screen "Root screen" 800x480, template "Main"
   Button "Button_1" at 525,223 size 98x74; TextOff 'Text'
      on Click: InvertBit("V1_CMD_Start_M")
      Visibility <- "Logick_hand"
   Button "Button_2" at 409,219 size 32x177; TextOff 'Text'
      on Click: InvertBit("V2_CMD_Start_M")
      Visibility <- "Logick_hand"
   Button "Button_6" at 252,16 size 115x197; TextOff 'Text'
      on Click: InvertBit("T1_CMD_Start_M")
      Visibility <- "Logick_hand"
   Button "Button_12" at 225,303 size 168x65; TextOff 'Text'
      on Click: InvertBit("T3_CMD_Start_M")
      Visibility <- "Logick_hand"
   Button "Button_13" at 453,307 size 192x61; TextOff 'Text'
      on Click: InvertBit("T2_CMD_Start_M")
      Visibility <- "Logick_hand"
   Button "Button_3" at 269,227 size 85x72; TextOff 'Text'
      on Click: InvertBit("V3_CMD_Start_M")
      Visibility <- "Logick_hand"
   Button "Button_4" at 175,16 size 73x115; TextOff 'Text'
      on Click: InvertBit("T0_CMD_Start_M")
      Visibility <- "Logick_hand"
   Rectangle "Rectangle_25" at 421,348 size 10x46
      Visibility <- "Valves_DB_V2_Status"
   IOField "I/O field_1" at 262,49 size 96x32; FormatPattern 999.9
      ProcessValue <- "AOx_DB_SP_CF_SP_M"
      Appearance <- "AOx_DB_SP_CF_CMD_Hand"
   Rectangle "Rectangle_17" at 130,379 size 23x10
      Appearance <- "T3_Box_Ready_Signal"
   Rectangle "Rectangle_18" at 133,375 size 17x5
      Appearance <- "T3_Box_Ready_Signal"
   Rectangle "Rectangle_19" at 302,379 size 23x10
      Appearance <- "T2_Box_Ready_Signal"
   Rectangle "Rectangle_20" at 305,375 size 17x5
      Appearance <- "T2_Box_Ready_Signal"
   Rectangle "Rectangle_21" at 451,379 size 23x10
      Appearance <- "T1_Box_ready_Signal"
   Rectangle "Rectangle_22" at 454,375 size 17x5
      Appearance <- "T1_Box_ready_Signal"
   Button "Button_15" at 31,168 size 178x54; TextOff 'Пропустить'
      on Click: SetBit("T3V3W3_DB_Skip_box")
      Appearance <- "main_screens"
   Rectangle "Rectangle_2" at 252,16 size 115x230
      Appearance <- "T1_Status"
   Rectangle "Rectangle_3" at 14,253 size 199x115
      Appearance <- "T4_Status"
   Rectangle "Rectangle_4" at 225,253 size 168x115
      Appearance <- "T3_Status"
   Rectangle "Rectangle_5" at 406,253 size 239x115
      Appearance <- "T2_Status"
   Rectangle "Rectangle_6" at 421,247 size 10x46
      Visibility <- "Valves_DB_V2_Status"
   Rectangle "Rectangle_7" at 421,326 size 10x46
      Visibility <- "Valves_DB_V2_Status"
   Rectangle "Rectangle_8" at 568,243 size 10x38
      Visibility <- "Valves_DB_V1_Status"
   Rectangle "Rectangle_9" at 542,280 size 62x10
      Visibility <- "Valves_DB_V1_Status"
   TextField "Text field_2" at 612,341 size 49x28; Text 'T2'
   TextField "Text field_3" at 361,340 size 49x28; Text 'T3'
   TextField "Text field_4" at 178,341 size 49x28; Text 'T4'
   Rectangle "Rectangle_10" at 421,223 size 10x46
      Visibility <- "Valves_DB_V2_Status"
   Rectangle "Rectangle_11" at 421,348 size 10x46
      Visibility <- "Valves_DB_V2_Status"
   Rectangle "Rectangle_12" at 569,223 size 10x38
      Visibility <- "Valves_DB_V1_Status"
   Rectangle "Rectangle_13" at 543,260 size 62x10
      Visibility <- "Valves_DB_V1_Status"
   TextField "Text field_7" at 433,227 size 43x23; Text 'V2'
   TextField "Text field_8" at 579,227 size 43x23; Text 'V1'
   Button "Button_8" at 376,17 size 175x60; TextOff 'Авто'
      on Release: SetBit("Logic_DB_Start_weight")
      Appearance <- "Logic_DB_Start_weight"
   Button "Button_9" at 376,85 size 175x60; TextOff 'Стоп'
      on Release: ResetBit("Logic_DB_Start_weight")
   Button "Button_10" at 376,153 size 175x60; TextOff 'Ручной'; Authorization "Operator"
      on Click: InvertBit("Logick_hand")
      Appearance <- "Logick_hand"
   IOField "I/O field_4" at 556,17 size 175x60; FormatPattern 99.9
      ProcessValue <- "T3V3W3_DB_SetPoints_SP"
   TextField "Text field_17" at 588,84 size 112x62; Text 'кг'
   Rectangle "Rectangle_24" at 421,223 size 10x46
      Visibility <- "Valves_DB_V2_Status"
   Rectangle "Rectangle_26" at 421,223 size 10x46
      Visibility <- "Valves_DB_V2_Status"
   Rectangle "Rectangle_27" at 421,348 size 10x46
      Visibility <- "Valves_DB_V2_Status"
   Rectangle "Rectangle_28" at 569,224 size 10x38
      Visibility <- "Valves_DB_V1_Status"
   Rectangle "Rectangle_29" at 543,260 size 62x10
      Visibility <- "Valves_DB_V1_Status"
   Rectangle "Rectangle_30" at 569,224 size 10x38
      Visibility <- "Valves_DB_V1_Status"
   Rectangle "Rectangle_31" at 543,260 size 62x10
      Visibility <- "Valves_DB_V1_Status"
   TextField "Text field_11" at 20,48 size 135x52; Text 'Тунель охлаждения'
   IOField "I/O field_2" at 556,153 size 175x60; FormatPattern s99.9
      ProcessValue <- "T3V3W3_DB_LocalVar_SP_loaded"
   Rectangle "Rectangle_32" at 175,16 size 73x115
      Appearance <- "T0_Status"
   TextField "Text field_1" at 189,15 size 49x28; Text 'T0'
   TextField "Text field_12" at 285,13 size 49x28; Text 'T1'
   Circle "Circle_1" at 270,220 size 82x82
      Appearance <- "V3_Status"
   Button "Button_11" at 14,253 size 199x115; TextOff 'Text'
      on Click: InvertBit("T4_CMD_Start_M")
      Visibility <- "Logick_hand"
   TextField "Text field_13" at 298,250 size 43x23; Text 'V3'
   Group "Group" at 130,375 size 23x30
   Group "Group_1" at 302,375 size 23x30
   Group "Group_2" at 451,375 size 23x30
   TextField "Template_Text field_1" at 525,59 size 27x15; Text 'F1'
   TextField "Template_Text field_2" at 525,127 size 27x15; Text 'F2'
   Button "Button_21" at 556,153 size 173x61; TextOff 'Установка нуля'; TextList "Hand"
      on Click: InvertBit("T3V3W3_DB_Reset_weight")
      ProcessValue <- "ODT1_CMD_Hand"
      Visibility <- "Logic_DB_Start_weight"
   Button "Button_5" at 14,415 size 211x58; TextOff 'Обзор'
      on Click: ActivateScreen("Root screen", 0); SetTag("main_screens", 0)
      Appearance <- "main_screens"
   Button "Button_14" at 264,415 size 211x58; TextOff 'Вес'
      on Click: ActivateScreen("weight", 0); SetTag("main_screens", 1)
      Appearance <- "main_screens"
   Button "Button_7" at 513,415 size 211x58; TextOff 'Статистика'
      on Click: ActivateScreen("statistic", 0); SetTag("main_screens", 2); SetTag("stat_view", 0)
      Appearance <- "main_screens"
   Rectangle "Rectangle_33" at 5,269 size 732x211
      Visibility <- "T3V3W3_DB_Reload"
   Rectangle "Rectangle_23" at 32,134 size 175x115
      Visibility <- "Any_Hand"
      Appearance <- "Any_Hand"
   TextField "Text field_5" at 142,306 size 455x58; Text 'Некорректный вес.'
      Visibility <- "T3V3W3_DB_Reload"
   Button "Button_16" at 193,388 size 345x75; TextOff 'Продолжить'
      on Click: SetBit("Reset_All")
      Visibility <- "T3V3W3_DB_Reload"
   TextField "Text field_10" at 36,140 size 169x99; Text 'Внимание! Часть устройств в ручном режиме. Корректная работа невозможна.'
      Visibility <- "Any_Hand"
      Appearance <- "Any_Hand"
   Rectangle "Rectangle_34" at 5,268 size 732x211
      Visibility <- "T3V3W3_DB_No_box"
   Button "Button_20" at 197,387 size 345x75; TextOff 'Продолжить'
      on Click: ResetBit("T3V3W3_DB_No_box")
      Visibility <- "T3V3W3_DB_No_box"
   TextField "Text field_6" at 216,305 size 311x58; Text 'Нет коробки.'
      Visibility <- "T3V3W3_DB_No_box"

screen "Conveyors_0" 800x480, template "Main"
   Rectangle "Rectangle_2" at 127,146 size 416x126
      Appearance <- "T3_CMD_Sim"
   GraphicIOField "Graphic I/O field_1" at 134,182 size 43x85; PictureList "Motor"
      ProcessValue <- "T3_Status"
   Button "Button_10" at 213,180 size 90x22; TextOff 'Авто'; TextList "Hand"
      on Click: InvertBit("T3_CMD_Hand")
      Appearance <- "T3_CMD_Hand"
      ProcessValue <- "T3_CMD_Hand"
   Button "Button_12" at 258,202 size 45x22; TextOff 'Выкл'
      on Click: ResetBit("T3_CMD_Start_M")
   Button "Button_14" at 213,225 size 90x20; TextOff 'Сервис'
      on Click: InvertBit("T3_CMD_Service")
      Appearance <- "T3_CMD_Service"
   Button "Button_15" at 213,202 size 45x22; TextOff 'Вкл'
      on Click: SetBit("T3_CMD_Start_M")
      Appearance <- "T3_CMD_Start_M"
   TextField "Text field_6" at 133,151 size 171x26; Text 'Конвеер 3'
   TextField "Text field_7" at 310,151 size 99x18; Text 'Ожидание ОС, с'
   GraphicView "Graphic view_2" at 180,181 size 25x25; Picture "z2use_3"
      Visibility <- "T3_CMD_Hand"
   GraphicView "Graphic view_3" at 180,213 size 25x25; Picture "force"
      Visibility <- "T3_CMD_Force"
   GraphicView "Graphic view_4" at 180,242 size 25x25; Picture "service"
      Visibility <- "T3_CMD_Service"
   TextField "Text field_8" at 436,170 size 20x18; Text 'QF'
   TextField "Text field_9" at 436,195 size 21x18; Text 'KM'
   TextField "Text field_11" at 436,221 size 44x18; Text 'Service'
   TextField "Text field_16" at 436,247 size 41x18; Text 'Termo'
   TextField "Text field_17" at 416,149 size 120x22; Text 'Использовать:'
   Button "Button_16" at 478,171 size 60x20; TextOff 'Text'; PictureList "ON_OFF"; Authorization "Operator"
      on Click: InvertBit("T3_Use_QF")
      ProcessValue <- "T3_Use_QF"
   Button "Button_17" at 478,195 size 60x20; TextOff 'Text'; Authorization "Operator"; PictureList "ON_OFF"
      on Click: InvertBit("T3_Use_KM")
      ProcessValue <- "T3_Use_KM"
   Button "Button_18" at 478,219 size 60x20; TextOff 'Text'; Authorization "Operator"; PictureList "ON_OFF"
      on Click: InvertBit("T3_Use_Serivce")
      ProcessValue <- "T3_Use_Serivce"
   Button "Button_19" at 478,244 size 60x20; TextOff 'Text'; Authorization "Operator"; PictureList "ON_OFF"
      on Click: InvertBit("T3_Use_Termo")
      ProcessValue <- "T3_Use_Termo"
   Button "Button_20" at 416,170 size 20x20; TextOff 'Text'; PictureList "ok"; Authorization "Operator"
      ProcessValue <- "T3_FB_QF"
   Button "Button_23" at 416,194 size 20x20; TextOff 'Text'; Authorization "Operator"; PictureList "ok"
      ProcessValue <- "T3_FB_KM"
   Button "Button_28" at 416,219 size 20x20; TextOff 'Text'; Authorization "Operator"; PictureList "ok"
      ProcessValue <- "T3_Use_Serivce"
   Button "Button_31" at 416,244 size 20x20; TextOff 'Text'; Authorization "Operator"; PictureList "ok"
      ProcessValue <- "T3_FB_Termo"
   TextField "Text field_18" at 323,226 size 79x18; Text 'Наработка, ч'
   TextField "Text field_19" at 309,173 size 37x18; Text 'Старт'
   IOField "I/O field_1" at 348,171 size 30x20; FormatPattern 99
      ProcessValue <- "T3_Wait_On_SP"
   IOField "I/O field_2" at 348,194 size 30x20; FormatPattern 99
      ProcessValue <- "T3_Wait_Off_SP"
   TextField "Text field_20" at 309,194 size 32x18; Text 'Стоп'
   IOField "I/O field_3" at 378,171 size 30x20; FormatPattern 99
      ProcessValue <- "T3_Wait_On_Now"
   IOField "I/O field_4" at 378,194 size 30x20; FormatPattern 99
      ProcessValue <- "T3_Wait_Off_Now"
   IOField "I/O field_6" at 313,244 size 98x20; FormatPattern 9999999999
      ProcessValue <- "T3_Res_h"
   Button "Button_32" at 213,245 size 90x20; TextOff 'Force'
      on Click: InvertBit("T3_CMD_Force")
      Appearance <- "T3_CMD_Force"
   Rectangle "Rectangle_3" at 127,285 size 416x126
      Appearance <- "T4_CMD_Sim"
   GraphicIOField "Graphic I/O field_3" at 134,321 size 43x85; PictureList "Motor"
      ProcessValue <- "T4_Status"
   Button "Button_33" at 213,319 size 90x22; TextOff 'Авто'; TextList "Hand"
      on Click: InvertBit("T4_CMD_Hand")
      Appearance <- "T4_CMD_Hand"
      ProcessValue <- "T4_CMD_Hand"
   Button "Button_34" at 258,341 size 45x22; TextOff 'Выкл'
      on Click: ResetBit("T4_CMD_Start_M")
   Button "Button_35" at 213,364 size 90x20; TextOff 'Сервис'
      on Click: InvertBit("T4_CMD_Service")
      Appearance <- "T4_CMD_Service"
   Button "Button_36" at 213,341 size 45x22; TextOff 'Вкл'
      on Click: SetBit("T4_CMD_Start_M")
      Appearance <- "T4_CMD_Start_M"
   TextField "Text field_21" at 133,290 size 171x26; Text 'Конвеер 4'
   TextField "Text field_22" at 310,290 size 99x18; Text 'Ожидание ОС, с'
   GraphicView "Graphic view_5" at 180,320 size 25x25; Picture "z2use_3"
      Visibility <- "T4_CMD_Hand"
   GraphicView "Graphic view_6" at 180,352 size 25x25; Picture "force"
      Visibility <- "T4_CMD_Force"
   GraphicView "Graphic view_7" at 180,381 size 25x25; Picture "service"
      Visibility <- "T4_CMD_Service"
   TextField "Text field_23" at 436,309 size 20x18; Text 'QF'
   TextField "Text field_24" at 436,334 size 21x18; Text 'KM'
   TextField "Text field_25" at 436,360 size 44x18; Text 'Service'
   TextField "Text field_26" at 436,386 size 41x18; Text 'Termo'
   TextField "Text field_27" at 416,288 size 120x22; Text 'Использовать:'
   Button "Button_37" at 478,310 size 60x20; TextOff 'Text'; PictureList "ON_OFF"; Authorization "Operator"
      on Click: InvertBit("T4_Use_QF")
      ProcessValue <- "T4_Use_QF"
   Button "Button_38" at 478,334 size 60x20; TextOff 'Text'; Authorization "Operator"; PictureList "ON_OFF"
      on Click: InvertBit("T4_Use_KM")
      ProcessValue <- "T4_Use_KM"
   Button "Button_39" at 478,358 size 60x20; TextOff 'Text'; Authorization "Operator"; PictureList "ON_OFF"
      on Click: InvertBit("T4_Use_Serivce")
      ProcessValue <- "T4_Use_Serivce"
   Button "Button_40" at 478,383 size 60x20; TextOff 'Text'; Authorization "Operator"; PictureList "ON_OFF"
      on Click: InvertBit("T4_Use_Termo")
      ProcessValue <- "T4_Use_Termo"
   Button "Button_41" at 416,309 size 20x20; TextOff 'Text'; PictureList "ok"; Authorization "Operator"
      ProcessValue <- "T4_FB_QF"
   Button "Button_42" at 416,333 size 20x20; TextOff 'Text'; Authorization "Operator"; PictureList "ok"
      ProcessValue <- "T4_FB_KM"
   Button "Button_43" at 416,358 size 20x20; TextOff 'Text'; Authorization "Operator"; PictureList "ok"
      ProcessValue <- "T4_Use_Serivce"
   Button "Button_44" at 416,383 size 20x20; TextOff 'Text'; Authorization "Operator"; PictureList "ok"
      ProcessValue <- "T4_FB_Termo"
   TextField "Text field_28" at 323,365 size 79x18; Text 'Наработка, ч'
   TextField "Text field_29" at 309,312 size 37x18; Text 'Старт'
   IOField "I/O field_7" at 348,310 size 30x20; FormatPattern 99
      ProcessValue <- "T4_Wait_On_SP"
   IOField "I/O field_8" at 348,333 size 30x20; FormatPattern 99
      ProcessValue <- "T4_Wait_Off_SP"
   TextField "Text field_30" at 309,333 size 32x18; Text 'Стоп'
   IOField "I/O field_9" at 378,310 size 30x20; FormatPattern 99
      ProcessValue <- "T4_Wait_On_Now"
   IOField "I/O field_10" at 378,333 size 30x20; FormatPattern 99
      ProcessValue <- "T4_Wait_Off_Now"
   IOField "I/O field_11" at 313,383 size 98x20; FormatPattern 9999999999
      ProcessValue <- "T4_Res_h"
   Button "Button_45" at 213,384 size 90x20; TextOff 'Force'
      on Click: InvertBit("T4_CMD_Force")
      Appearance <- "T4_CMD_Force"
   Rectangle "Rectangle_1" at 127,7 size 416x126
      Appearance <- "T2_CMD_Sim"
   GraphicIOField "Graphic I/O field_2" at 134,43 size 43x85; PictureList "Motor"
      ProcessValue <- "T2_Status"
   Button "Button_7" at 213,41 size 90x22; TextOff 'Авто'; TextList "Hand"
      on Click: InvertBit("T2_CMD_Hand")
      Appearance <- "T2_CMD_Hand"
      ProcessValue <- "T2_CMD_Hand"
   Button "Button_8" at 258,63 size 45x22; TextOff 'Выкл'
      on Click: ResetBit("T2_CMD_Start_M")
   Button "Button_9" at 213,86 size 90x20; TextOff 'Сервис'
      on Click: InvertBit("T2_CMD_Service")
      Appearance <- "T2_CMD_Service"
   Button "Button_13" at 213,63 size 45x22; TextOff 'Вкл'
      on Click: SetBit("T2_CMD_Start_M")
      Appearance <- "T2_CMD_Start_M"
   TextField "Text field_13" at 133,12 size 171x26; Text 'Конвеер 2'
   TextField "Text field_15" at 310,12 size 99x18; Text 'Ожидание ОС, с'
   GraphicView "Graphic view_1" at 180,42 size 25x25; Picture "z2use_3"
      Visibility <- "T2_CMD_Hand"
   GraphicView "Graphic view_8" at 180,74 size 25x25; Picture "force"
      Visibility <- "T2_CMD_Force"
   GraphicView "Graphic view_11" at 180,103 size 25x25; Picture "service"
      Visibility <- "T2_CMD_Service"
   TextField "Text field_3" at 436,31 size 20x18; Text 'QF'
   TextField "Text field_10" at 436,56 size 21x18; Text 'KM'
   TextField "Text field_12" at 436,82 size 44x18; Text 'Service'
   TextField "Text field_14" at 436,108 size 41x18; Text 'Termo'
   TextField "Text field_4" at 416,10 size 120x22; Text 'Использовать:'
   Button "Button_21" at 478,32 size 60x20; TextOff 'Text'; Authorization "Operator"; PictureList "ON_OFF"
      on Click: InvertBit("T2_Use_QF")
      ProcessValue <- "T2_Use_QF"
   Button "Button_22" at 478,56 size 60x20; TextOff 'Text'; PictureList "ON_OFF"; Authorization "Operator"
      on Click: InvertBit("T2_Use_KM")
      ProcessValue <- "T2_Use_KM"
   Button "Button_24" at 478,80 size 60x20; TextOff 'Text'; PictureList "ON_OFF"; Authorization "Operator"
      on Click: InvertBit("T2_Use_Serivce")
      ProcessValue <- "T2_Use_Serivce"
   Button "Button_25" at 478,105 size 60x20; TextOff 'Text'; PictureList "ON_OFF"; Authorization "Operator"
      on Click: InvertBit("T2_Use_Termo")
      ProcessValue <- "T2_Use_Termo"
   Button "Button_26" at 416,31 size 20x20; TextOff 'Text'; Authorization "Operator"; PictureList "ok"
      ProcessValue <- "T2_FB_QF"
   Button "Button_27" at 416,55 size 20x20; TextOff 'Text'; PictureList "ok"; Authorization "Operator"
      ProcessValue <- "T2_FB_KM"
   Button "Button_29" at 416,80 size 20x20; TextOff 'Text'; PictureList "ok"; Authorization "Operator"
      ProcessValue <- "T2_Use_Serivce"
   Button "Button_30" at 416,105 size 20x20; TextOff 'Text'; PictureList "ok"; Authorization "Operator"
      ProcessValue <- "T2_FB_Termo"
   TextField "Text field_1" at 323,87 size 79x18; Text 'Наработка, ч'
   TextField "Text field_2" at 309,34 size 37x18; Text 'Старт'
   IOField "I/O field_5" at 348,32 size 30x20; FormatPattern 99
      ProcessValue <- "T2_Wait_On_SP"
   IOField "I/O field_12" at 348,55 size 30x20; FormatPattern 99
      ProcessValue <- "T2_Wait_Off_SP"
   TextField "Text field_5" at 309,55 size 32x18; Text 'Стоп'
   IOField "I/O field_13" at 378,32 size 30x20; FormatPattern 99
      ProcessValue <- "T2_Wait_On_Now"
   IOField "I/O field_14" at 378,55 size 30x20; FormatPattern 99
      ProcessValue <- "T2_Wait_Off_Now"
   IOField "I/O field_16" at 313,105 size 98x20; FormatPattern 9999999999
      ProcessValue <- "T2_Res_h"
   Button "Button_11" at 213,106 size 90x20; TextOff 'Force'
      on Click: InvertBit("T2_CMD_Force")
      Appearance <- "T2_CMD_Force"
   Button "Button_1" at 7,5 size 96x32; TextOff 'Коробки'; Authorization "Admin"
      on Release: ActivateScreen("Conveyors_0", 0); SetTag("settings", 1)
      Appearance <- "settings"
   Button "Button_2" at 7,51 size 96x32; TextOff 'Шоколад'; Authorization "Admin"
      on Release: ActivateScreen("Conveyors_1", 0); SetTag("settings", 2)
      Appearance <- "settings"
   Button "Button_3" at 7,98 size 96x32; TextOff 'Клапана'; Authorization "Admin"
      on Release: SetTag("settings", 3); ActivateScreen("Valve", 0)
      Appearance <- "settings"
   Button "Button_4" at 7,145 size 96x32; TextOff 'DI 1'; Authorization "Admin"
      on Release: SetTag("settings", 4); ActivateScreen("DI_1", 0)
      Appearance <- "settings"
   Button "Button_5" at 7,191 size 96x32; TextOff 'DI 2'; Authorization "Admin"
      on Release: SetTag("settings", 5); ActivateScreen("DI_2", 0)
      Appearance <- "settings"
   Button "Button_6" at 7,238 size 96x32; TextOff 'DO'; Authorization "Admin"
      on Release: SetTag("settings", 6); ActivateScreen("DO", 0)
      Appearance <- "settings"
   Button "Button_46" at 7,285 size 96x32; TextOff 'Весы'; Authorization "Admin"
      on Press: ActivateScreen("0.0.0_Service_Quick_Start", 0)
      Appearance <- "settings"

screen "Conveyors_1" 800x480, template "Main"
   Rectangle "Rectangle_2" at 127,5 size 416x126
      Appearance <- "T0_CMD_Sim"
   GraphicIOField "Graphic I/O field_1" at 134,41 size 43x85; PictureList "Motor"
      ProcessValue <- "T0_Status"
   Button "Button_10" at 213,39 size 90x22; TextOff 'Авто'; TextList "Hand"
      on Click: InvertBit("T0_CMD_Hand")
      Appearance <- "T0_CMD_Hand"
      ProcessValue <- "T0_CMD_Hand"
   Button "Button_12" at 258,61 size 45x22; TextOff 'Выкл'
      on Click: ResetBit("T0_CMD_Start_M")
   Button "Button_14" at 213,84 size 90x20; TextOff 'Сервис'
      on Click: InvertBit("T0_CMD_Service")
      Appearance <- "T0_CMD_Service"
   Button "Button_15" at 213,61 size 45x22; TextOff 'Вкл'
      on Click: SetBit("T0_CMD_Start_M")
      Appearance <- "T0_CMD_Start_M"
   TextField "Text field_6" at 133,10 size 171x26; Text 'Конвеер 0'
   TextField "Text field_7" at 310,10 size 99x18; Text 'Ожидание ОС, с'
   GraphicView "Graphic view_2" at 180,40 size 25x25; Picture "z2use_3"
      Visibility <- "T0_CMD_Hand"
   GraphicView "Graphic view_3" at 180,72 size 25x25; Picture "force"
      Visibility <- "T0_CMD_Force"
   GraphicView "Graphic view_4" at 180,101 size 25x25; Picture "service"
      Visibility <- "T0_CMD_Service"
   TextField "Text field_8" at 436,29 size 20x18; Text 'QF'
   TextField "Text field_9" at 436,54 size 21x18; Text 'KM'
   TextField "Text field_11" at 436,80 size 44x18; Text 'Service'
   TextField "Text field_16" at 436,106 size 41x18; Text 'Termo'
   TextField "Text field_17" at 416,8 size 120x22; Text 'Использовать:'
   Button "Button_16" at 478,30 size 60x20; TextOff 'Text'; PictureList "ON_OFF"; Authorization "Operator"
      on Click: InvertBit("T0_Use_QF")
      ProcessValue <- "T0_Use_QF"
   Button "Button_17" at 478,54 size 60x20; TextOff 'Text'; Authorization "Operator"; PictureList "ON_OFF"
      on Click: InvertBit("T0_Use_KM")
      ProcessValue <- "T0_Use_KM"
   Button "Button_18" at 478,78 size 60x20; TextOff 'Text'; Authorization "Operator"; PictureList "ON_OFF"
      on Click: InvertBit("T0_Use_Serivce")
      ProcessValue <- "T0_Use_Serivce"
   Button "Button_19" at 478,103 size 60x20; TextOff 'Text'; Authorization "Operator"; PictureList "ON_OFF"
      on Click: InvertBit("T0_Use_Termo")
      ProcessValue <- "T0_Use_Termo"
   Button "Button_20" at 416,29 size 20x20; TextOff 'Text'; PictureList "ok"; Authorization "Operator"
      ProcessValue <- "T0_FB_QF"
   Button "Button_23" at 416,53 size 20x20; TextOff 'Text'; Authorization "Operator"; PictureList "ok"
      ProcessValue <- "T0_FB_KM"
   Button "Button_28" at 416,78 size 20x20; TextOff 'Text'; Authorization "Operator"; PictureList "ok"
      ProcessValue <- "T0_Use_Serivce"
   Button "Button_31" at 416,103 size 20x20; TextOff 'Text'; Authorization "Operator"; PictureList "ok"
      ProcessValue <- "T0_FB_Termo"
   TextField "Text field_18" at 323,85 size 79x18; Text 'Наработка, ч'
   TextField "Text field_19" at 309,32 size 37x18; Text 'Старт'
   IOField "I/O field_1" at 348,30 size 30x20; FormatPattern 99
      ProcessValue <- "T0_Wait_On_SP"
   IOField "I/O field_2" at 348,53 size 30x20; FormatPattern 99
      ProcessValue <- "T0_Wait_Off_SP"
   TextField "Text field_20" at 309,53 size 32x18; Text 'Стоп'
   IOField "I/O field_3" at 378,30 size 30x20; FormatPattern 99
      ProcessValue <- "T0_Wait_On_Now"
   IOField "I/O field_4" at 378,53 size 30x20; FormatPattern 99
      ProcessValue <- "T0_Wait_Off_Now"
   IOField "I/O field_6" at 313,103 size 98x20; FormatPattern 9999999999
      ProcessValue <- "T0_Res_h"
   Button "Button_32" at 213,104 size 90x20; TextOff 'Force'
      on Click: InvertBit("T0_CMD_Force")
      Appearance <- "T0_CMD_Force"
   Rectangle "Rectangle_1" at 127,139 size 416x126
      Appearance <- "T1_CMD_Sim"
   GraphicIOField "Graphic I/O field_2" at 134,175 size 43x85; PictureList "Motor"
      ProcessValue <- "T1_Status"
   Button "Button_7" at 213,173 size 90x22; TextOff 'Авто'; TextList "Hand"
      on Click: InvertBit("T1_CMD_Hand")
      Appearance <- "T1_CMD_Hand"
      ProcessValue <- "T1_CMD_Hand"
   Button "Button_8" at 258,195 size 45x22; TextOff 'Выкл'
      on Click: ResetBit("T1_CMD_Start_M")
   Button "Button_9" at 213,218 size 90x20; TextOff 'Сервис'
      on Click: InvertBit("T1_CMD_Service")
      Appearance <- "T1_CMD_Service"
   Button "Button_13" at 213,195 size 45x22; TextOff 'Вкл'
      on Click: SetBit("T1_CMD_Start_M")
      Appearance <- "T1_CMD_Start_M"
   TextField "Text field_13" at 133,144 size 171x26; Text 'Конвеер 1'
   TextField "Text field_15" at 310,144 size 99x18; Text 'Ожидание ОС, с'
   GraphicView "Graphic view_1" at 180,174 size 25x25; Picture "z2use_3"
      Visibility <- "T1_CMD_Hand"
   GraphicView "Graphic view_8" at 180,206 size 25x25; Picture "force"
      Visibility <- "T1_CMD_Force"
   GraphicView "Graphic view_11" at 180,235 size 25x25; Picture "service"
      Visibility <- "T1_CMD_Service"
   TextField "Text field_3" at 436,163 size 20x18; Text 'QF'
   TextField "Text field_10" at 436,188 size 21x18; Text 'KM'
   TextField "Text field_12" at 436,214 size 44x18; Text 'Service'
   TextField "Text field_14" at 436,240 size 41x18; Text 'Termo'
   TextField "Text field_4" at 416,142 size 120x22; Text 'Использовать:'
   Button "Button_21" at 478,164 size 60x20; TextOff 'Text'; PictureList "ON_OFF"; Authorization "Operator"
      on Click: InvertBit("T1_Use_QF")
      ProcessValue <- "T1_Use_QF"
   Button "Button_22" at 478,188 size 60x20; TextOff 'Text'; Authorization "Operator"; PictureList "ON_OFF"
      on Click: InvertBit("T1_Use_KM")
      ProcessValue <- "T1_Use_KM"
   Button "Button_24" at 478,212 size 60x20; TextOff 'Text'; Authorization "Operator"; PictureList "ON_OFF"
      on Click: InvertBit("T1_Use_Serivce")
      ProcessValue <- "T1_Use_Serivce"
   Button "Button_25" at 478,237 size 60x20; TextOff 'Text'; Authorization "Operator"; PictureList "ON_OFF"
      on Click: InvertBit("T1_Use_Termo")
      ProcessValue <- "T1_Use_Termo"
   Button "Button_26" at 416,163 size 20x20; TextOff 'Text'; PictureList "ok"; Authorization "Operator"
      ProcessValue <- "T1_FB_QF"
   Button "Button_27" at 416,187 size 20x20; TextOff 'Text'; Authorization "Operator"; PictureList "ok"
      ProcessValue <- "T1_FB_KM"
   Button "Button_29" at 416,212 size 20x20; TextOff 'Text'; Authorization "Operator"; PictureList "ok"
      ProcessValue <- "T1_Use_Serivce"
   Button "Button_30" at 416,237 size 20x20; TextOff 'Text'; Authorization "Operator"; PictureList "ok"
      ProcessValue <- "T1_FB_Termo"
   TextField "Text field_1" at 323,219 size 79x18; Text 'Наработка, ч'
   TextField "Text field_2" at 309,166 size 37x18; Text 'Старт'
   IOField "I/O field_5" at 348,164 size 30x20; FormatPattern 99
      ProcessValue <- "T1_Wait_On_SP"
   IOField "I/O field_12" at 348,187 size 30x20; FormatPattern 99
      ProcessValue <- "T1_Wait_Off_SP"
   TextField "Text field_5" at 309,187 size 32x18; Text 'Стоп'
   IOField "I/O field_13" at 378,164 size 30x20; FormatPattern 99
      ProcessValue <- "T1_Wait_On_Now"
   IOField "I/O field_14" at 378,187 size 30x20; FormatPattern 99
      ProcessValue <- "T1_Wait_Off_Now"
   IOField "I/O field_16" at 313,237 size 98x20; FormatPattern 9999999999
      ProcessValue <- "T1_Res_h"
   Button "Button_11" at 213,238 size 90x20; TextOff 'Force'
      on Click: InvertBit("T1_CMD_Force")
      Appearance <- "T1_CMD_Force"
   Button "Button_1" at 7,5 size 96x32; TextOff 'Коробки'; Authorization "Admin"
      on Release: ActivateScreen("Conveyors_0", 0); SetTag("settings", 1)
      Appearance <- "settings"
   Button "Button_2" at 7,51 size 96x32; TextOff 'Шоколад'; Authorization "Admin"
      on Release: ActivateScreen("Conveyors_1", 0); SetTag("settings", 2)
      Appearance <- "settings"
   Button "Button_3" at 7,98 size 96x32; TextOff 'Клапана'; Authorization "Admin"
      on Release: SetTag("settings", 3); ActivateScreen("Valve", 0)
      Appearance <- "settings"
   Button "Button_4" at 7,145 size 96x32; TextOff 'DI 1'; Authorization "Admin"
      on Release: SetTag("settings", 4); ActivateScreen("DI_1", 0)
      Appearance <- "settings"
   Button "Button_5" at 7,191 size 96x32; TextOff 'DI 2'; Authorization "Admin"
      on Release: SetTag("settings", 5); ActivateScreen("DI_2", 0)
      Appearance <- "settings"
   Button "Button_6" at 7,238 size 96x32; TextOff 'DO'; Authorization "Admin"
      on Release: SetTag("settings", 6); ActivateScreen("DO", 0)
      Appearance <- "settings"
   Button "Button_33" at 7,285 size 96x32; TextOff 'Весы'; Authorization "Admin"
      on Press: ActivateScreen("0.0.0_Service_Quick_Start", 0)
      Appearance <- "settings"

screen "Valve" 800x480, template "Main"
   Rectangle "Rectangle_1" at 127,7 size 521x126
      Appearance <- "V1_CMD_Sim"
   Button "Button_7" at 213,41 size 90x22; TextOff 'Авто'; TextList "Hand"
      on Click: InvertBit("V1_CMD_Hand")
      Appearance <- "V1_CMD_Hand"
      ProcessValue <- "V1_CMD_Hand"
   Button "Button_8" at 258,63 size 45x22; TextOff 'Выкл'
      on Click: ResetBit("V1_CMD_Start_M")
   Button "Button_9" at 213,86 size 90x20; TextOff 'Сервис'
      on Click: InvertBit("V1_CMD_Service")
      Appearance <- "V1_CMD_Service"
   Button "Button_13" at 213,63 size 45x22; TextOff 'Вкл'
      on Click: SetBit("V1_CMD_Start_M")
      Appearance <- "V1_CMD_Start_M"
   TextField "Text field_13" at 133,12 size 171x26; Text 'Клапан 1'
   TextField "Text field_15" at 310,12 size 99x18; Text 'Ожидание ОС, с'
   GraphicView "Graphic view_1" at 180,42 size 25x25; Picture "z2use_3"
      Visibility <- "V1_CMD_Hand"
   GraphicView "Graphic view_8" at 180,74 size 25x25; Picture "force"
      Visibility <- "V1_CMD_Force"
   GraphicView "Graphic view_11" at 180,103 size 25x25; Picture "service"
      Visibility <- "V1_CMD_Service"
   TextField "Text field_3" at 535,31 size 31x18; Text 'Air'
   TextField "Text field_10" at 535,56 size 35x18; Text 'Open'
   TextField "Text field_12" at 535,107 size 44x18; Text 'Service'
   TextField "Text field_4" at 515,10 size 120x22; Text 'Использовать:'
   Button "Button_21" at 577,32 size 60x20; TextOff 'Text'; Authorization "Operator"; PictureList "ON_OFF"
      on Click: InvertBit("V1_Use_QF")
      ProcessValue <- "V1_Use_QF"
   Button "Button_22" at 577,56 size 60x20; TextOff 'Text'; PictureList "ON_OFF"; Authorization "Operator"
      on Click: InvertBit("V1_Use_Open")
      ProcessValue <- "V1_Use_Open"
   Button "Button_24" at 577,105 size 60x20; TextOff 'Text'; PictureList "ON_OFF"; Authorization "Operator"
      on Click: InvertBit("V1_Use_Serivce")
      ProcessValue <- "V1_Use_Serivce"
   Button "Button_26" at 515,31 size 20x20; TextOff 'Text'; Authorization "Operator"; PictureList "ok"
      ProcessValue <- "V1_FB_QF"
   Button "Button_27" at 515,55 size 20x20; TextOff 'Text'; PictureList "ok"; Authorization "Operator"
      ProcessValue <- "V1_FB_Open"
   Button "Button_29" at 515,105 size 20x20; TextOff 'Text'; PictureList "ok"; Authorization "Operator"
      ProcessValue <- "V1_FB_Service"
   TextField "Text field_1" at 323,87 size 79x18; Text 'Наработка, ч'
   TextField "Text field_2" at 309,34 size 37x18; Text 'Старт'
   IOField "I/O field_5" at 348,32 size 30x20; FormatPattern 99
      ProcessValue <- "V1_Wait_On_SP"
   IOField "I/O field_12" at 348,55 size 30x20; FormatPattern 99
      ProcessValue <- "V1_Wait_Off_SP"
   TextField "Text field_5" at 309,55 size 32x18; Text 'Стоп'
   IOField "I/O field_13" at 378,32 size 30x20; FormatPattern 99
      ProcessValue <- "V1_Wait_On_Now"
   IOField "I/O field_14" at 378,55 size 30x20; FormatPattern 99
      ProcessValue <- "V1_Wait_Off_Now"
   IOField "I/O field_16" at 313,105 size 98x20; FormatPattern 9999999999
      ProcessValue <- "V1_Res_h"
   Button "Button_11" at 213,106 size 90x20; TextOff 'Force'
      on Click: InvertBit("V1_CMD_Force")
      Appearance <- "V1_CMD_Force"
   GraphicIOField "Graphic I/O field_5" at 129,56 size 50x50; PictureList "Valve"
      ProcessValue <- "V1_Status"
   TextField "Text field_6" at 535,80 size 33x18; Text 'Close'
   Button "Button_10" at 577,80 size 60x20; TextOff 'Text'; Authorization "Operator"; PictureList "ON_OFF"
      on Click: InvertBit("V1_Use_Close")
      ProcessValue <- "V1_Use_Close"
   Button "Button_12" at 515,79 size 20x20; TextOff 'Text'; Authorization "Operator"; PictureList "ok"
      ProcessValue <- "V1_FB_Close"
   Rectangle "Rectangle_2" at 127,144 size 521x126
      Appearance <- "V2_CMD_Sim"
   Button "Button_14" at 213,178 size 90x22; TextOff 'Авто'; TextList "Hand"
      on Click: InvertBit("V2_CMD_Hand")
      Appearance <- "V2_CMD_Hand"
      ProcessValue <- "V2_CMD_Hand"
   Button "Button_15" at 258,200 size 45x22; TextOff 'Выкл'
      on Click: ResetBit("V2_CMD_Start_M")
   Button "Button_16" at 213,223 size 90x20; TextOff 'Сервис'
      on Click: InvertBit("V2_CMD_Service")
      Appearance <- "V2_CMD_Service"
   Button "Button_17" at 213,200 size 45x22; TextOff 'Вкл'
      on Click: SetBit("V2_CMD_Start_M")
      Appearance <- "V2_CMD_Start_M"
   TextField "Text field_7" at 133,149 size 171x26; Text 'Клапан 2'
   TextField "Text field_8" at 310,149 size 99x18; Text 'Ожидание ОС, с'
   GraphicView "Graphic view_2" at 180,179 size 25x25; Picture "z2use_3"
      Visibility <- "V2_CMD_Hand"
   GraphicView "Graphic view_3" at 180,211 size 25x25; Picture "force"
      Visibility <- "V2_CMD_Force"
   GraphicView "Graphic view_4" at 180,240 size 25x25; Picture "service"
      Visibility <- "V2_CMD_Service"
   TextField "Text field_9" at 535,168 size 31x18; Text 'Air'
   TextField "Text field_11" at 535,193 size 35x18; Text 'Open'
   TextField "Text field_14" at 535,244 size 44x18; Text 'Service'
   TextField "Text field_16" at 515,147 size 120x22; Text 'Использовать:'
   Button "Button_18" at 577,169 size 60x20; TextOff 'Text'; PictureList "ON_OFF"; Authorization "Operator"
      on Click: InvertBit("V2_Use_QF")
      ProcessValue <- "V2_Use_QF"
   Button "Button_19" at 577,193 size 60x20; TextOff 'Text'; Authorization "Operator"; PictureList "ON_OFF"
      on Click: InvertBit("V2_Use_Open")
      ProcessValue <- "V2_Use_Open"
   Button "Button_20" at 577,242 size 60x20; TextOff 'Text'; Authorization "Operator"; PictureList "ON_OFF"
      on Click: InvertBit("V2_Use_Serivce")
      ProcessValue <- "V2_Use_Serivce"
   Button "Button_23" at 515,168 size 20x20; TextOff 'Text'; PictureList "ok"; Authorization "Operator"
      ProcessValue <- "V2_FB_QF"
   Button "Button_25" at 515,192 size 20x20; TextOff 'Text'; Authorization "Operator"; PictureList "ok"
      ProcessValue <- "V2_FB_Open"
   Button "Button_28" at 515,242 size 20x20; TextOff 'Text'; Authorization "Operator"; PictureList "ok"
      ProcessValue <- "V2_FB_Service"
   TextField "Text field_17" at 323,225 size 79x18; Text 'Наработка, ч'
   TextField "Text field_18" at 309,171 size 37x18; Text 'Старт'
   IOField "I/O field_1" at 348,169 size 30x20; FormatPattern 99
      ProcessValue <- "V2_Wait_On_SP"
   IOField "I/O field_2" at 348,192 size 30x20; FormatPattern 99
      ProcessValue <- "V2_Wait_Off_SP"
   TextField "Text field_19" at 309,192 size 32x18; Text 'Стоп'
   IOField "I/O field_3" at 378,169 size 30x20; FormatPattern 99
      ProcessValue <- "V2_Wait_On_Now"
   IOField "I/O field_4" at 378,192 size 30x20; FormatPattern 99
      ProcessValue <- "V2_Wait_Off_Now"
   IOField "I/O field_6" at 313,243 size 98x20; FormatPattern 9999999999
      ProcessValue <- "V2_Res_h"
   Button "Button_30" at 213,243 size 90x20; TextOff 'Force'
      on Click: InvertBit("V2_CMD_Force")
      Appearance <- "V2_CMD_Force"
   GraphicIOField "Graphic I/O field_1" at 129,193 size 50x50; PictureList "Valve"
      ProcessValue <- "Valves_DB_V2_Status"
   TextField "Text field_20" at 535,217 size 33x18; Text 'Close'
   Button "Button_31" at 577,217 size 60x20; TextOff 'Text'; PictureList "ON_OFF"; Authorization "Operator"
      on Click: InvertBit("V2_Use_Close")
      ProcessValue <- "V2_Use_Close"
   Button "Button_32" at 515,216 size 20x20; TextOff 'Text'; PictureList "ok"; Authorization "Operator"
      ProcessValue <- "V2_FB_Close"
   Rectangle "Rectangle_3" at 127,279 size 521x126
      Appearance <- "V3_CMD_Sim"
   Button "Button_33" at 213,313 size 90x22; TextOff 'Авто'; TextList "Hand"
      on Click: InvertBit("V3_CMD_Hand")
      Appearance <- "V3_CMD_Hand"
      ProcessValue <- "V3_CMD_Hand"
   Button "Button_34" at 258,335 size 45x22; TextOff 'Выкл'
      on Click: ResetBit("V3_CMD_Start_M")
   Button "Button_35" at 213,358 size 90x20; TextOff 'Сервис'
      on Click: InvertBit("V3_CMD_Service")
      Appearance <- "V3_CMD_Service"
   Button "Button_36" at 213,335 size 45x22; TextOff 'Вкл'
      on Click: SetBit("V3_CMD_Start_M")
      Appearance <- "V3_CMD_Start_M"
   TextField "Text field_21" at 133,284 size 171x26; Text 'Клапан 3'
   TextField "Text field_22" at 310,284 size 99x18; Text 'Ожидание ОС, с'
   GraphicView "Graphic view_5" at 180,314 size 25x25; Picture "z2use_3"
      Visibility <- "V3_CMD_Hand"
   GraphicView "Graphic view_6" at 180,346 size 25x25; Picture "force"
      Visibility <- "V3_CMD_Force"
   GraphicView "Graphic view_7" at 180,375 size 25x25; Picture "service"
      Visibility <- "V3_CMD_Service"
   TextField "Text field_23" at 535,303 size 31x18; Text 'Air'
   TextField "Text field_24" at 535,328 size 35x18; Text 'Open'
   TextField "Text field_25" at 535,379 size 44x18; Text 'Service'
   TextField "Text field_26" at 515,282 size 120x22; Text 'Использовать:'
   Button "Button_37" at 577,304 size 60x20; TextOff 'Text'; PictureList "ON_OFF"; Authorization "Operator"
      on Click: InvertBit("V3_Use_QF")
      ProcessValue <- "V3_Use_QF"
   Button "Button_38" at 577,328 size 60x20; TextOff 'Text'; Authorization "Operator"; PictureList "ON_OFF"
      on Click: InvertBit("V3_Use_Open")
      ProcessValue <- "V3_Use_Open"
   Button "Button_39" at 577,377 size 60x20; TextOff 'Text'; Authorization "Operator"; PictureList "ON_OFF"
      on Click: InvertBit("V3_Use_Serivce")
      ProcessValue <- "V3_Use_Serivce"
   Button "Button_40" at 515,303 size 20x20; TextOff 'Text'; PictureList "ok"; Authorization "Operator"
      ProcessValue <- "V3_FB_QF"
   Button "Button_41" at 515,327 size 20x20; TextOff 'Text'; Authorization "Operator"; PictureList "ok"
      ProcessValue <- "V3_FB_Open"
   Button "Button_42" at 515,377 size 20x20; TextOff 'Text'; Authorization "Operator"; PictureList "ok"
      ProcessValue <- "V3_FB_Service"
   TextField "Text field_27" at 323,361 size 79x18; Text 'Наработка, ч'
   TextField "Text field_28" at 309,306 size 37x18; Text 'Старт'
   IOField "I/O field_7" at 348,304 size 30x20; FormatPattern 99
      ProcessValue <- "V3_Wait_On_SP"
   IOField "I/O field_8" at 348,327 size 30x20; FormatPattern 99
      ProcessValue <- "V3_Wait_Off_SP"
   TextField "Text field_29" at 309,327 size 32x18; Text 'Стоп'
   IOField "I/O field_9" at 378,304 size 30x20; FormatPattern 99
      ProcessValue <- "V3_Wait_On_Now"
   IOField "I/O field_10" at 378,327 size 30x20; FormatPattern 99
      ProcessValue <- "V3_Wait_Off_Now"
   IOField "I/O field_11" at 313,379 size 98x20; FormatPattern 9999999999
      ProcessValue <- "V3_Res_h"
   Button "Button_43" at 213,378 size 90x20; TextOff 'Force'
      on Click: InvertBit("V3_CMD_Force")
      Appearance <- "V3_CMD_Force"
   GraphicIOField "Graphic I/O field_2" at 129,328 size 50x50; PictureList "Valve"
      ProcessValue <- "V3_Status"
   TextField "Text field_30" at 535,352 size 33x18; Text 'Close'
   Button "Button_44" at 577,352 size 60x20; TextOff 'Text'; PictureList "ON_OFF"; Authorization "Operator"
      on Click: InvertBit("V3_Use_Close")
      ProcessValue <- "V3_Use_Close"
   Button "Button_45" at 515,351 size 20x20; TextOff 'Text'; PictureList "ok"; Authorization "Operator"
      ProcessValue <- "V3_FB_Close"
   TextField "Text field_31" at 427,12 size 60x18; Text 'Задержка'
   TextField "Text field_32" at 438,34 size 37x18; Text 'Старт'
   IOField "I/O field_15" at 423,55 size 35x20; FormatPattern 99.9
      ProcessValue <- "Valves_DB_V1_Delay_On_SP"
   IOField "I/O field_17" at 423,105 size 35x20; FormatPattern 99.9
      ProcessValue <- "Valves_DB_V1_Delay_Off_SP"
   TextField "Text field_33" at 441,84 size 32x18; Text 'Стоп'
   IOField "I/O field_18" at 461,55 size 35x20; FormatPattern 99.9
      ProcessValue <- "Valves_DB_V1_Delay_On_Now"
   IOField "I/O field_19" at 461,105 size 35x20; FormatPattern 99.9
      ProcessValue <- "Valves_DB_V1_Delay_Off_Now"
   TextField "Text field_34" at 428,149 size 60x18; Text 'Задержка'
   TextField "Text field_35" at 439,171 size 37x18; Text 'Старт'
   IOField "I/O field_20" at 424,192 size 35x20; FormatPattern 99.9
      ProcessValue <- "Valves_DB_V2_Delay_On_SP"
   IOField "I/O field_21" at 424,242 size 35x20; FormatPattern 99.9
      ProcessValue <- "Valves_DB_V2_Delay_Off_SP"
   TextField "Text field_36" at 442,221 size 32x18; Text 'Стоп'
   IOField "I/O field_22" at 462,192 size 35x20; FormatPattern 99.9
      ProcessValue <- "Valves_DB_V2_Delay_On_Now"
   IOField "I/O field_23" at 462,242 size 35x20; FormatPattern 99.9
      ProcessValue <- "Valves_DB_V2_Delay_Off_Now"
   TextField "Text field_37" at 429,286 size 60x18; Text 'Задержка'
   TextField "Text field_38" at 440,308 size 37x18; Text 'Старт'
   IOField "I/O field_24" at 425,329 size 35x20; FormatPattern 99.9
      ProcessValue <- "Valves_DB_V3_Delay_On_SP"
   IOField "I/O field_25" at 425,379 size 35x20; FormatPattern 99.9
      ProcessValue <- "Valves_DB_V3_Delay_Off_SP"
   TextField "Text field_39" at 443,358 size 32x18; Text 'Стоп'
   IOField "I/O field_26" at 463,329 size 35x20; FormatPattern 99.9
      ProcessValue <- "Valves_DB_V3_Delay_On_Now"
   IOField "I/O field_27" at 463,379 size 35x20; FormatPattern 99.9
      ProcessValue <- "Valves_DB_V3_Delay_Off_Now"
   Button "Button_1" at 7,5 size 96x32; TextOff 'Коробки'; Authorization "Admin"
      on Release: ActivateScreen("Conveyors_0", 0); SetTag("settings", 1)
      Appearance <- "settings"
   Button "Button_2" at 7,51 size 96x32; TextOff 'Шоколад'; Authorization "Admin"
      on Release: ActivateScreen("Conveyors_1", 0); SetTag("settings", 2)
      Appearance <- "settings"
   Button "Button_3" at 7,98 size 96x32; TextOff 'Клапана'; Authorization "Admin"
      on Release: SetTag("settings", 3); ActivateScreen("Valve", 0)
      Appearance <- "settings"
   Button "Button_4" at 7,145 size 96x32; TextOff 'DI 1'; Authorization "Admin"
      on Release: SetTag("settings", 4); ActivateScreen("DI_1", 0)
      Appearance <- "settings"
   Button "Button_5" at 7,191 size 96x32; TextOff 'DI 2'; Authorization "Admin"
      on Release: SetTag("settings", 5); ActivateScreen("DI_2", 0)
      Appearance <- "settings"
   Button "Button_6" at 7,238 size 96x32; TextOff 'DO'; Authorization "Admin"
      on Release: SetTag("settings", 6); ActivateScreen("DO", 0)
      Appearance <- "settings"
   Button "Button_46" at 7,285 size 96x32; TextOff 'Весы'; Authorization "Admin"
      on Press: ActivateScreen("0.0.0_Service_Quick_Start", 0)
      Appearance <- "settings"

screen "DI_1" 800x480, template "Main"
   TextField "Text field_23" at 437,187 size 45x22; Text 'I 1.3'
   TextField "Text field_24" at 482,187 size 93x22; Text 'Т3 Коробка'
   Circle "Circle_23" at 437,210 size 22x22
      Appearance <- "T3_Box_Ready_Input"
   Circle "Circle_24" at 460,210 size 22x22
      Appearance <- "T3_Box_Ready_Signal"
   Button "Button_51" at 604,188 size 59x44; TextOff 'Авто'; TextList "Hand"
      on Click: InvertBit("T3_Box_Ready_Hand")
      Appearance <- "T3_Box_Ready_Hand"
      ProcessValue <- "T3_Box_Ready_Hand"
   Button "Button_52" at 546,210 size 49x22; TextOff 'Выкл'
      on Click: ResetBit("T3_Box_Ready_Start_M")
   Button "Button_53" at 490,210 size 47x22; TextOff 'Вкл'
      on Click: SetBit("T3_Box_Ready_Start_M")
      Appearance <- "T3_Box_Ready_Start_M"
   IOField "I/O field_23" at 666,210 size 23x22; FormatPattern 99
      ProcessValue <- "T3_Box_Ready_Filter_On_SP"
   IOField "I/O field_24" at 689,210 size 23x22; FormatPattern 99
      ProcessValue <- "T3_Box_Ready_Filter_Off_SP"
   Button "Button_54" at 666,187 size 46x20; TextOff 'Inv'
      on Click: InvertBit("T3_Box_Ready_Inverse")
      Appearance <- "T3_Box_Ready_Inverse"
   TextField "Text field_21" at 437,128 size 45x22; Text 'I 1.2'
   TextField "Text field_22" at 482,128 size 93x22; Text 'Т2 Коробка'
   Circle "Circle_21" at 437,151 size 22x22
      Appearance <- "T2_Box_Ready_Input"
   Circle "Circle_22" at 460,151 size 22x22
      Appearance <- "T2_Box_Ready_Signal"
   Button "Button_47" at 604,129 size 59x44; TextOff 'Авто'; TextList "Hand"
      on Click: InvertBit("T2_Box_Ready_Hand")
      Appearance <- "T2_Box_Ready_Hand"
      ProcessValue <- "T2_Box_Ready_Hand"
   Button "Button_48" at 546,151 size 49x22; TextOff 'Выкл'
      on Click: ResetBit("T2_Box_Ready_Start_M")
   Button "Button_49" at 490,151 size 47x22; TextOff 'Вкл'
      on Click: SetBit("T2_Box_Ready_Start_M")
      Appearance <- "T2_Box_Ready_Start_M"
   IOField "I/O field_21" at 666,151 size 23x22; FormatPattern 99
      ProcessValue <- "T2_Box_Ready_Filter_On_SP"
   IOField "I/O field_22" at 689,151 size 23x22; FormatPattern 99
      ProcessValue <- "T2_Box_Ready_Filter_Off_SP"
   Button "Button_50" at 666,128 size 46x20; TextOff 'Inv'
      on Click: InvertBit("T2_Box_Ready_Inverse")
      Appearance <- "T2_Box_Ready_Inverse"
   TextField "Text field_19" at 437,69 size 45x22; Text 'I 1.1'
   TextField "Text field_20" at 482,69 size 93x22; Text 'T1 Коробка'
   Circle "Circle_19" at 437,92 size 22x22
      Appearance <- "T1_Box_ready_Input"
   Circle "Circle_20" at 460,92 size 22x22
      Appearance <- "T1_Box_ready_Signal"
   Button "Button_43" at 604,70 size 59x44; TextOff 'Авто'; TextList "Hand"
      on Click: InvertBit("T1_Box_ready_Hand")
      Appearance <- "T1_Box_ready_Hand"
      ProcessValue <- "T1_Box_ready_Hand"
   Button "Button_44" at 546,92 size 49x22; TextOff 'Выкл'
      on Click: ResetBit("T1_Box_ready_Start_M")
   Button "Button_45" at 490,92 size 47x22; TextOff 'Вкл'
      on Click: SetBit("T1_Box_ready_Start_M")
      Appearance <- "T1_Box_ready_Start_M"
   IOField "I/O field_19" at 666,92 size 23x22; FormatPattern 99
      ProcessValue <- "T1_Box_ready_Filter_On_SP"
   IOField "I/O field_20" at 689,92 size 23x22; FormatPattern 99
      ProcessValue <- "T1_Box_ready_Filter_Off_SP"
   Button "Button_46" at 666,69 size 46x20; TextOff 'Inv'
      on Click: InvertBit("T1_Box_ready_Inverse")
      Appearance <- "T1_Box_ready_Inverse"
   TextField "Text field_17" at 437,10 size 45x22; Text 'I 1.0'
   TextField "Text field_18" at 482,10 size 118x22; Text 'Конвеер Т3 QF'
   Circle "Circle_17" at 437,33 size 22x22
      Appearance <- "T3_QF_Input"
   Circle "Circle_18" at 460,33 size 22x22
      Appearance <- "T3_QF_Signal"
   Button "Button_39" at 604,11 size 59x44; TextOff 'Авто'; TextList "Hand"
      on Click: InvertBit("T3_QF_Hand")
      Appearance <- "T3_QF_Hand"
      ProcessValue <- "T3_QF_Hand"
   Button "Button_40" at 546,33 size 49x22; TextOff 'Выкл'
      on Click: ResetBit("T3_QF_Start_M")
   Button "Button_41" at 490,33 size 47x22; TextOff 'Вкл'
      on Click: SetBit("T3_QF_Start_M")
      Appearance <- "T3_QF_Start_M"
   IOField "I/O field_17" at 666,33 size 23x22; FormatPattern 99
      ProcessValue <- "T3_QF_Filter_On_SP"
   IOField "I/O field_18" at 689,33 size 23x22; FormatPattern 99
      ProcessValue <- "T3_QF_Filter_Off_SP"
   Button "Button_42" at 666,10 size 46x20; TextOff 'Inv'
      on Click: InvertBit("T3_QF_Inverse")
      Appearance <- "T3_QF_Inverse"
   TextField "Text field_7" at 131,187 size 45x22; Text 'I 0.3'
   TextField "Text field_8" at 176,187 size 104x22; Text 'Питание 24В'
   Circle "Circle_7" at 131,210 size 22x22
      Appearance <- "Voltage_24V_Ok_Input"
   Circle "Circle_8" at 154,210 size 22x22
      Appearance <- "Voltage_24V_Ok_Signal"
   Button "Button_19" at 298,188 size 59x44; TextOff 'Авто'; TextList "Hand"
      on Click: InvertBit("Voltage_24V_Ok_Hand")
      Appearance <- "Voltage_24V_Ok_Hand"
      ProcessValue <- "Voltage_24V_Ok_Hand"
   Button "Button_20" at 240,210 size 49x22; TextOff 'Выкл'
      on Click: ResetBit("Voltage_24V_Ok_Start_M")
   Button "Button_21" at 184,210 size 47x22; TextOff 'Вкл'
      on Click: SetBit("Voltage_24V_Ok_Start_M")
      Appearance <- "Voltage_24V_Ok_Start_M"
   IOField "I/O field_5" at 360,210 size 23x22; FormatPattern 99
      ProcessValue <- "Voltage_24V_Ok_Filter_On_SP"
   IOField "I/O field_8" at 383,210 size 23x22; FormatPattern 99
      ProcessValue <- "Voltage_24V_Ok_Filter_Off_SP"
   Button "Button_22" at 360,187 size 46x20; TextOff 'Inv'
      on Click: InvertBit("Voltage_24V_Ok_Inverse")
      Appearance <- "Voltage_24V_Ok_Inverse"
   TextField "Text field_5" at 131,128 size 45x22; Text 'I 0.2'
   TextField "Text field_6" at 176,128 size 97x22; Text 'Питание DO'
   Circle "Circle_5" at 131,151 size 22x22
      Appearance <- "Voltage_DO_Ok_Input"
   Circle "Circle_6" at 154,151 size 22x22
      Appearance <- "Voltage_DO_Ok_Signal"
   Button "Button_15" at 298,129 size 59x44; TextOff 'Авто'; TextList "Hand"
      on Click: InvertBit("Voltage_DO_Ok_Hand")
      Appearance <- "Voltage_DO_Ok_Hand"
      ProcessValue <- "Voltage_DO_Ok_Hand"
   Button "Button_16" at 240,151 size 49x22; TextOff 'Выкл'
      on Click: ResetBit("Voltage_DO_Ok_Start_M")
   Button "Button_17" at 184,151 size 47x22; TextOff 'Вкл'
      on Click: SetBit("Voltage_DO_Ok_Start_M")
      Appearance <- "Voltage_DO_Ok_Start_M"
   IOField "I/O field_3" at 360,151 size 23x22; FormatPattern 99
      ProcessValue <- "Voltage_DO_Ok_Filter_On_SP"
   IOField "I/O field_4" at 383,151 size 23x22; FormatPattern 99
      ProcessValue <- "Voltage_DO_Ok_Filter_Off_SP"
   Button "Button_18" at 360,128 size 46x20; TextOff 'Inv'
      on Click: InvertBit("Voltage_DO_Ok_Inverse")
      Appearance <- "Voltage_DO_Ok_Inverse"
   TextField "Text field_3" at 131,69 size 45x22; Text 'I 0.1'
   TextField "Text field_4" at 176,69 size 92x22; Text 'Питание DI'
   Circle "Circle_3" at 131,92 size 22x22
      Appearance <- "Voltage_DI_Ok_Input"
   Circle "Circle_4" at 154,92 size 22x22
      Appearance <- "Voltage_DI_Ok_Signal"
   Button "Button_10" at 298,70 size 59x44; TextOff 'Авто'; TextList "Hand"
      on Click: InvertBit("Voltage_DI_Ok_Hand")
      Appearance <- "Voltage_DI_Ok_Hand"
      ProcessValue <- "Voltage_DI_Ok_Hand"
   Button "Button_11" at 240,92 size 49x22; TextOff 'Выкл'
      on Click: ResetBit("Voltage_DI_Ok_Start_M")
   Button "Button_13" at 184,92 size 47x22; TextOff 'Вкл'
      on Click: SetBit("Voltage_DI_Ok_Start_M")
      Appearance <- "Voltage_DI_Ok_Start_M"
   IOField "I/O field_1" at 360,92 size 23x22; FormatPattern 99
      ProcessValue <- "Voltage_DI_Ok_Filter_On_SP"
   IOField "I/O field_2" at 383,92 size 23x22; FormatPattern 99
      ProcessValue <- "Voltage_DI_Ok_Filter_Off_SP"
   Button "Button_14" at 360,69 size 46x20; TextOff 'Inv'
      on Click: InvertBit("Voltage_DI_Ok_Inverse")
      Appearance <- "Voltage_DI_Ok_Inverse"
   TextField "Text field_1" at 131,10 size 45x22; Text 'I 0.0'
   TextField "Text field_2" at 176,10 size 105x22; Text 'Питание CPU'
   Circle "Circle_1" at 131,33 size 22x22
      Appearance <- "Voltage_CPU_Ok_Input"
   Circle "Circle_2" at 154,33 size 22x22
      Appearance <- "Voltage_CPU_Ok_Signal"
   Button "Button_7" at 298,11 size 59x44; TextOff 'Авто'; TextList "Hand"
      on Click: InvertBit("Voltage_CPU_Ok_Hand")
      Appearance <- "Voltage_CPU_Ok_Hand"
      ProcessValue <- "Voltage_CPU_Ok_Hand"
   Button "Button_8" at 240,33 size 49x22; TextOff 'Выкл'
      on Click: ResetBit("Voltage_CPU_Ok_Start_M")
   Button "Button_12" at 184,33 size 47x22; TextOff 'Вкл'
      on Click: SetBit("Voltage_CPU_Ok_Start_M")
      Appearance <- "Voltage_CPU_Ok_Start_M"
   IOField "I/O field_6" at 360,33 size 23x22; FormatPattern 99
      ProcessValue <- "Voltage_CPU_Ok_Filter_On_SP"
   IOField "I/O field_7" at 383,33 size 23x22; FormatPattern 99
      ProcessValue <- "Voltage_CPU_Ok_Filter_Off_SP"
   Button "Button_9" at 360,10 size 46x20; TextOff 'Inv'
      on Click: InvertBit("Voltage_CPU_Ok_Inverse")
      Appearance <- "Voltage_CPU_Ok_Inverse"
   TextField "Text field_25" at 437,247 size 45x22; Text 'I 1.4'
   TextField "Text field_26" at 482,247 size 114x22; Text 'Давлен. возд.'
   Circle "Circle_25" at 437,270 size 22x22
      Appearance <- "Air_pressure_Ok_Input"
   Circle "Circle_26" at 460,270 size 22x22
      Appearance <- "Air_pressure_Ok_Signal"
   Button "Button_55" at 604,248 size 59x44; TextOff 'Авто'; TextList "Hand"
      on Click: InvertBit("Air_pressure_Ok_Hand")
      Appearance <- "Air_pressure_Ok_Hand"
      ProcessValue <- "Air_pressure_Ok_Hand"
   Button "Button_56" at 546,270 size 49x22; TextOff 'Выкл'
      on Click: ResetBit("Air_pressure_Ok_Start_M")
   Button "Button_57" at 490,270 size 47x22; TextOff 'Вкл'
      on Click: SetBit("Air_pressure_Ok_Start_M")
      Appearance <- "Air_pressure_Ok_Start_M"
   IOField "I/O field_25" at 666,270 size 23x22; FormatPattern 99
      ProcessValue <- "Air_pressure_Ok_Filter_On_SP"
   IOField "I/O field_26" at 689,270 size 23x22; FormatPattern 99
      ProcessValue <- "Air_pressure_Ok_Filter_Off_SP"
   Button "Button_58" at 666,247 size 46x20; TextOff 'Inv'
      on Click: InvertBit("Air_pressure_Ok_Inverse")
      Appearance <- "Air_pressure_Ok_Inverse"
   TextField "Text field_15" at 131,425 size 45x22; Text 'I 0.7'
   TextField "Text field_16" at 176,425 size 118x22; Text 'Конвеер Т2 QF'
   Circle "Circle_15" at 131,448 size 22x22
      Appearance <- "T2_QF_Input"
   Circle "Circle_16" at 154,448 size 22x22
      Appearance <- "T2_QF_Signal"
   Button "Button_35" at 298,426 size 59x44; TextOff 'Авто'; TextList "Hand"
      on Click: InvertBit("T2_QF_Hand")
      Appearance <- "T2_QF_Hand"
      ProcessValue <- "T2_QF_Hand"
   Button "Button_36" at 240,448 size 49x22; TextOff 'Выкл'
      on Click: ResetBit("T2_QF_Start_M")
   Button "Button_37" at 184,448 size 47x22; TextOff 'Вкл'
      on Click: SetBit("T2_QF_Start_M")
      Appearance <- "T2_QF_Start_M"
   IOField "I/O field_15" at 360,448 size 23x22; FormatPattern 99
      ProcessValue <- "T2_QF_Filter_On_SP"
   IOField "I/O field_16" at 383,448 size 23x22; FormatPattern 99
      ProcessValue <- "T2_QF_Filter_Off_SP"
   Button "Button_38" at 360,425 size 46x20; TextOff 'Inv'
      on Click: InvertBit("T2_QF_Inverse")
      Appearance <- "T2_QF_Inverse"
   TextField "Text field_13" at 131,365 size 45x22; Text 'I 0.6'
   TextField "Text field_14" at 176,365 size 118x22; Text 'Конвеер Т1 QF'
   Circle "Circle_13" at 131,388 size 22x22
      Appearance <- "T1_QF_Input"
   Circle "Circle_14" at 154,388 size 22x22
      Appearance <- "T1_QF_Signal"
   Button "Button_31" at 298,366 size 59x44; TextOff 'Авто'; TextList "Hand"
      on Click: InvertBit("T1_QF_Hand")
      Appearance <- "T1_QF_Hand"
      ProcessValue <- "T1_QF_Hand"
   Button "Button_32" at 240,388 size 49x22; TextOff 'Выкл'
      on Click: ResetBit("T1_QF_Start_M")
   Button "Button_33" at 184,388 size 47x22; TextOff 'Вкл'
      on Click: SetBit("T1_QF_Start_M")
      Appearance <- "T1_QF_Start_M"
   IOField "I/O field_13" at 360,388 size 23x22; FormatPattern 99
      ProcessValue <- "T1_QF_Filter_On_SP"
   IOField "I/O field_14" at 383,388 size 23x22; FormatPattern 99
      ProcessValue <- "T1_QF_Filter_Off_SP"
   Button "Button_34" at 360,365 size 46x20; TextOff 'Inv'
      on Click: InvertBit("T1_QF_Inverse")
      Appearance <- "T1_QF_Inverse"
   TextField "Text field_11" at 131,306 size 45x22; Text 'I 0.5'
   TextField "Text field_12" at 176,306 size 114x22; Text 'Cold tunnel QF'
   Circle "Circle_11" at 131,329 size 22x22
      Appearance <- "Cold_tunnel_QF_Input"
   Circle "Circle_12" at 154,329 size 22x22
      Appearance <- "Cold_tunnel_QF_Signal"
   Button "Button_27" at 298,307 size 59x44; TextOff 'Авто'; TextList "Hand"
      on Click: InvertBit("Cold_tunnel_QF_Hand")
      Appearance <- "Cold_tunnel_QF_Hand"
      ProcessValue <- "Cold_tunnel_QF_Hand"
   Button "Button_28" at 240,329 size 49x22; TextOff 'Выкл'
      on Click: ResetBit("Cold_tunnel_QF_Start_M")
   Button "Button_29" at 184,329 size 47x22; TextOff 'Вкл'
      on Click: SetBit("Cold_tunnel_QF_Start_M")
      Appearance <- "Cold_tunnel_QF_Start_M"
   IOField "I/O field_11" at 360,329 size 23x22; FormatPattern 99
      ProcessValue <- "Cold_tunnel_QF_Filter_On_SP"
   IOField "I/O field_12" at 383,329 size 23x22; FormatPattern 99
      ProcessValue <- "Cold_tunnel_QF_Filter_Off_SP"
   Button "Button_30" at 360,306 size 46x20; TextOff 'Inv'
      on Click: InvertBit("Cold_tunnel_QF_Inverse")
      Appearance <- "Cold_tunnel_QF_Inverse"
   TextField "Text field_9" at 131,247 size 45x22; Text 'I 0.4'
   TextField "Text field_10" at 176,247 size 111x22; Text 'Безопасность'
   Circle "Circle_9" at 131,270 size 22x22
      Appearance <- "Safety_Ok_Input"
   Circle "Circle_10" at 154,270 size 22x22
      Appearance <- "Safety_Ok_Signal"
   Button "Button_23" at 298,248 size 59x44; TextOff 'Авто'; TextList "Hand"
      on Click: InvertBit("Safety_Ok_Hand")
      Appearance <- "Safety_Ok_Hand"
      ProcessValue <- "Safety_Ok_Hand"
   Button "Button_24" at 240,270 size 49x22; TextOff 'Выкл'
      on Click: ResetBit("Safety_Ok_Start_M")
   Button "Button_25" at 184,270 size 47x22; TextOff 'Вкл'
      on Click: SetBit("Safety_Ok_Start_M")
      Appearance <- "Safety_Ok_Start_M"
   IOField "I/O field_9" at 360,270 size 23x22; FormatPattern 99
      ProcessValue <- "Safety_Ok_Filter_On_SP"
   IOField "I/O field_10" at 383,270 size 23x22; FormatPattern 99
      ProcessValue <- "Safety_Ok_Filter_Off_SP"
   Button "Button_26" at 360,247 size 46x20; TextOff 'Inv'
      on Click: InvertBit("Safety_Ok_Inverse")
      Appearance <- "Safety_Ok_Inverse"
   Button "Button_1" at 7,5 size 96x32; TextOff 'Коробки'; Authorization "Admin"
      on Release: ActivateScreen("Conveyors_0", 0); SetTag("settings", 1)
      Appearance <- "settings"
   Button "Button_2" at 7,51 size 96x32; TextOff 'Шоколад'; Authorization "Admin"
      on Release: ActivateScreen("Conveyors_1", 0); SetTag("settings", 2)
      Appearance <- "settings"
   Button "Button_3" at 7,98 size 96x32; TextOff 'Клапана'; Authorization "Admin"
      on Release: SetTag("settings", 3); ActivateScreen("Valve", 0)
      Appearance <- "settings"
   Button "Button_4" at 7,145 size 96x32; TextOff 'DI 1'; Authorization "Admin"
      on Release: SetTag("settings", 4); ActivateScreen("DI_1", 0)
      Appearance <- "settings"
   Button "Button_5" at 7,191 size 96x32; TextOff 'DI 2'; Authorization "Admin"
      on Release: SetTag("settings", 5); ActivateScreen("DI_2", 0)
      Appearance <- "settings"
   Button "Button_6" at 7,238 size 96x32; TextOff 'DO'; Authorization "Admin"
      on Release: SetTag("settings", 6); ActivateScreen("DO", 0)
      Appearance <- "settings"
   Button "Button_59" at 7,285 size 96x32; TextOff 'Весы'; Authorization "Admin"
      on Press: ActivateScreen("0.0.0_Service_Quick_Start", 0)
      Appearance <- "settings"

screen "DO" 800x480, template "Main"
   TextField "Text field_19" at 437,69 size 45x22; Text 'Q 2.1'
   TextField "Text field_20" at 482,69 size 48x22; Text 'Reset'
   Circle "Circle_19" at 437,92 size 22x22
      Appearance <- "Reset_Start_A"
   Circle "Circle_20" at 460,92 size 22x22
      Appearance <- "Reset_Q"
   Button "Button_52" at 604,70 size 59x44; TextOff 'Авто'; TextList "Hand"
      on Click: InvertBit("Reset_Hand")
      Appearance <- "Reset_Hand"
      ProcessValue <- "Reset_Hand"
   Button "Button_53" at 546,92 size 49x22; TextOff 'Выкл'
      on Click: ResetBit("Reset_Start_M")
   Button "Button_54" at 490,92 size 47x22; TextOff 'Вкл'
      on Click: SetBit("Reset_Start_M")
      Appearance <- "Reset_Start_M"
   Button "Button_55" at 666,69 size 46x20; TextOff 'Inv'
      on Click: InvertBit("Reset_Inverse")
      Appearance <- "Reset_Inverse"
   Button "Button_56" at 666,94 size 46x20; TextOff 'Sim'
      on Click: InvertBit("Reset_Simulation")
      Appearance <- "Reset_Simulation"
   TextField "Text field_17" at 437,10 size 45x22; Text 'Q 2.0'
   TextField "Text field_18" at 482,10 size 99x22; Text 'Reset safety'
   Circle "Circle_17" at 437,33 size 22x22
      Appearance <- "Reset_Safety_Start_A"
   Circle "Circle_18" at 460,33 size 22x22
      Appearance <- "Reset_Safety_Q"
   Button "Button_47" at 604,11 size 59x44; TextOff 'Авто'; TextList "Hand"
      on Click: InvertBit("Reset_Safety_Hand")
      Appearance <- "Reset_Safety_Hand"
      ProcessValue <- "Reset_Safety_Hand"
   Button "Button_48" at 546,33 size 49x22; TextOff 'Выкл'
      on Click: ResetBit("Reset_Safety_Start_M")
   Button "Button_49" at 490,33 size 47x22; TextOff 'Вкл'
      on Click: SetBit("Reset_Safety_Start_M")
      Appearance <- "Reset_Safety_Start_M"
   Button "Button_50" at 666,10 size 46x20; TextOff 'Inv'
      on Click: InvertBit("Reset_Safety_Inverse")
      Appearance <- "Reset_Safety_Inverse"
   Button "Button_51" at 666,35 size 46x20; TextOff 'Sim'
      on Click: InvertBit("Reset_Safety_Simulation")
      Appearance <- "Reset_Safety_Simulation"
   TextField "Text field_15" at 131,425 size 45x22; Text 'Q 0.7'
   TextField "Text field_16" at 176,425 size 119x22; Text 'Supply allowed'
   Circle "Circle_15" at 131,448 size 22x22
      Appearance <- "Supply_allowed_Start_A"
   Circle "Circle_16" at 154,448 size 22x22
      Appearance <- "Supply_allowed_Q"
   Button "Button_42" at 298,426 size 59x44; TextOff 'Авто'; TextList "Hand"
      on Click: InvertBit("Supply_allowed_Hand")
      Appearance <- "Supply_allowed_Hand"
      ProcessValue <- "Supply_allowed_Hand"
   Button "Button_43" at 240,448 size 49x22; TextOff 'Выкл'
      on Click: ResetBit("Supply_allowed_Start_M")
   Button "Button_44" at 184,448 size 47x22; TextOff 'Вкл'
      on Click: SetBit("Supply_allowed_Start_M")
      Appearance <- "Supply_allowed_Start_M"
   Button "Button_45" at 360,425 size 46x20; TextOff 'Inv'
      on Click: InvertBit("Supply_allowed_Inverse")
      Appearance <- "Supply_allowed_Inverse"
   Button "Button_46" at 360,450 size 46x20; TextOff 'Sim'
      on Click: InvertBit("Supply_allowed_Simulation")
      Appearance <- "Supply_allowed_Simulation"
   TextField "Text field_13" at 131,365 size 45x22; Text 'Q 0.6'
   TextField "Text field_14" at 176,365 size 63x22; Text 'K3 CMD'
   Circle "Circle_13" at 131,388 size 22x22
      Appearance <- "K3_CMD_Start_A"
   Circle "Circle_14" at 154,388 size 22x22
      Appearance <- "K3_CMD_Q"
   Button "Button_37" at 298,366 size 59x44; TextOff 'Авто'; TextList "Hand"
      on Click: InvertBit("K3_CMD_Hand")
      Appearance <- "K3_CMD_Hand"
      ProcessValue <- "K3_CMD_Hand"
   Button "Button_38" at 240,388 size 49x22; TextOff 'Выкл'
      on Click: ResetBit("K3_CMD_Start_M")
   Button "Button_39" at 184,388 size 47x22; TextOff 'Вкл'
      on Click: SetBit("K3_CMD_Start_M")
      Appearance <- "K3_CMD_Start_M"
   Button "Button_40" at 360,365 size 46x20; TextOff 'Inv'
      on Click: InvertBit("K3_CMD_Inverse")
      Appearance <- "K3_CMD_Inverse"
   Button "Button_41" at 360,390 size 46x20; TextOff 'Sim'
      on Click: InvertBit("K3_CMD_Simulation")
      Appearance <- "K3_CMD_Simulation"
   TextField "Text field_11" at 131,306 size 45x22; Text 'Q 0.5'
   TextField "Text field_12" at 176,306 size 63x22; Text 'K2 CMD'
   Circle "Circle_11" at 131,329 size 22x22
      Appearance <- "K2_CMD_Start_A"
   Circle "Circle_12" at 154,329 size 22x22
      Appearance <- "K2_CMD_Q"
   Button "Button_32" at 298,307 size 59x44; TextOff 'Авто'; TextList "Hand"
      on Click: InvertBit("K2_CMD_Hand")
      Appearance <- "K2_CMD_Hand"
      ProcessValue <- "K2_CMD_Hand"
   Button "Button_33" at 240,329 size 49x22; TextOff 'Выкл'
      on Click: ResetBit("K2_CMD_Start_M")
   Button "Button_34" at 184,329 size 47x22; TextOff 'Вкл'
      on Click: SetBit("K2_CMD_Start_M")
      Appearance <- "K2_CMD_Start_M"
   Button "Button_35" at 360,306 size 46x20; TextOff 'Inv'
      on Click: InvertBit("K2_CMD_Inverse")
      Appearance <- "K2_CMD_Inverse"
   Button "Button_36" at 360,331 size 46x20; TextOff 'Sim'
      on Click: InvertBit("K2_CMD_Simulation")
      Appearance <- "K2_CMD_Simulation"
   TextField "Text field_9" at 131,247 size 45x22; Text 'Q 0.4'
   TextField "Text field_10" at 176,247 size 63x22; Text 'K1 CMD'
   Circle "Circle_9" at 131,270 size 22x22
      Appearance <- "K1_CMD_Start_A"
   Circle "Circle_10" at 154,270 size 22x22
      Appearance <- "K1_CMD_Q"
   Button "Button_27" at 298,248 size 59x44; TextOff 'Авто'; TextList "Hand"
      on Click: InvertBit("K1_CMD_Hand")
      Appearance <- "K1_CMD_Hand"
      ProcessValue <- "K1_CMD_Hand"
   Button "Button_28" at 240,270 size 49x22; TextOff 'Выкл'
      on Click: ResetBit("K1_CMD_Start_M")
   Button "Button_29" at 184,270 size 47x22; TextOff 'Вкл'
      on Click: SetBit("K1_CMD_Start_M")
      Appearance <- "K1_CMD_Start_M"
   Button "Button_30" at 360,247 size 46x20; TextOff 'Inv'
      on Click: InvertBit("K1_CMD_Inverse")
      Appearance <- "K1_CMD_Inverse"
   Button "Button_31" at 360,272 size 46x20; TextOff 'Sim'
      on Click: InvertBit("K1_CMD_Simulation")
      Appearance <- "K1_CMD_Simulation"
   TextField "Text field_21" at 437,128 size 45x22; Text 'Q 2.1'
   TextField "Text field_22" at 482,128 size 50x22; Text 'Green'
   Circle "Circle_21" at 437,151 size 22x22
      Appearance <- "Green_Start_A"
   Circle "Circle_22" at 460,151 size 22x22
      Appearance <- "Green_Q"
   Button "Button_57" at 604,129 size 59x44; TextOff 'Авто'; TextList "Hand"
      on Click: InvertBit("Green_Hand")
      Appearance <- "Green_Hand"
      ProcessValue <- "Green_Hand"
   Button "Button_58" at 546,151 size 49x22; TextOff 'Выкл'
      on Click: ResetBit("Green_Start_M")
   Button "Button_59" at 490,151 size 47x22; TextOff 'Вкл'
      on Click: SetBit("Green_Start_M")
      Appearance <- "Green_Start_M"
   Button "Button_60" at 666,128 size 46x20; TextOff 'Inv'
      on Click: InvertBit("Green_Inverse")
      Appearance <- "Green_Inverse"
   Button "Button_61" at 666,153 size 46x20; TextOff 'Sim'
      on Click: InvertBit("Green_Simulation")
      Appearance <- "Green_Simulation"
   TextField "Text field_23" at 437,187 size 45x22; Text 'Q 2.1'
   TextField "Text field_24" at 482,187 size 38x22; Text 'Red'
   Circle "Circle_23" at 437,210 size 22x22
      Appearance <- "Red_Start_A"
   Circle "Circle_24" at 460,210 size 22x22
      Appearance <- "Red_Q"
   Button "Button_62" at 604,188 size 59x44; TextOff 'Авто'; TextList "Hand"
      on Click: InvertBit("Red_Hand")
      Appearance <- "Red_Hand"
      ProcessValue <- "Red_Hand"
   Button "Button_63" at 546,210 size 49x22; TextOff 'Выкл'
      on Click: ResetBit("Red_Start_M")
   Button "Button_64" at 490,210 size 47x22; TextOff 'Вкл'
      on Click: SetBit("Red_Start_M")
      Appearance <- "Red_Start_M"
   Button "Button_65" at 666,187 size 46x20; TextOff 'Inv'
      on Click: InvertBit("Red_Inverse")
      Appearance <- "Red_Inverse"
   Button "Button_66" at 666,212 size 46x20; TextOff 'Sim'
      on Click: InvertBit("Red_Simulation")
      Appearance <- "Red_Simulation"
   TextField "Text field_25" at 438,247 size 45x22; Text 'Q 2.1'
   TextField "Text field_26" at 483,247 size 38x22; Text 'Blue'
   Circle "Circle_25" at 438,270 size 22x22
      Appearance <- "Blue_Start_A"
   Circle "Circle_26" at 461,270 size 22x22
      Appearance <- "Blue_Q"
   Button "Button_67" at 605,248 size 59x44; TextOff 'Авто'; TextList "Hand"
      on Click: InvertBit("Blue_Hand")
      Appearance <- "Blue_Hand"
      ProcessValue <- "Blue_Hand"
   Button "Button_68" at 547,270 size 49x22; TextOff 'Выкл'
      on Click: ResetBit("Blue_Start_M")
   Button "Button_69" at 491,270 size 47x22; TextOff 'Вкл'
      on Click: SetBit("Blue_Start_M")
      Appearance <- "Blue_Start_M"
   Button "Button_70" at 667,247 size 46x20; TextOff 'Inv'
      on Click: InvertBit("Blue_Inverse")
      Appearance <- "Blue_Inverse"
   Button "Button_71" at 667,272 size 46x20; TextOff 'Sim'
      on Click: InvertBit("Blue_Simulation")
      Appearance <- "Blue_Simulation"
   TextField "Text field_27" at 438,307 size 45x22; Text 'Q 2.1'
   TextField "Text field_28" at 483,307 size 60x22; Text 'Orange'
   Circle "Circle_27" at 438,330 size 22x22
      Appearance <- "Orange_Start_A"
   Circle "Circle_28" at 461,330 size 22x22
      Appearance <- "Orange_Q"
   Button "Button_72" at 605,308 size 59x44; TextOff 'Авто'; TextList "Hand"
      on Click: InvertBit("Orange_Hand")
      Appearance <- "Orange_Hand"
      ProcessValue <- "Orange_Hand"
   Button "Button_73" at 547,330 size 49x22; TextOff 'Выкл'
      on Click: ResetBit("Orange_Start_M")
   Button "Button_74" at 491,330 size 47x22; TextOff 'Вкл'
      on Click: SetBit("Orange_Start_M")
      Appearance <- "Orange_Start_M"
   Button "Button_75" at 667,307 size 46x20; TextOff 'Inv'
      on Click: InvertBit("Orange_Inverse")
      Appearance <- "Orange_Inverse"
   Button "Button_76" at 667,332 size 46x20; TextOff 'Sim'
      on Click: InvertBit("Orange_Simulation")
      Appearance <- "Orange_Simulation"
   TextField "Text field_1" at 131,70 size 45x22; Text 'Q 2.1'
   TextField "Text field_2" at 176,70 size 62x22; Text 'T1 CMD'
   Circle "Circle_1" at 131,93 size 22x22
      Appearance <- "ODT1_CMD_Start_A"
   Circle "Circle_2" at 154,93 size 22x22
      Appearance <- "ODT1_CMD_Q"
   Button "Button_7" at 298,71 size 59x44; TextOff 'Авто'; TextList "Hand"
      on Click: InvertBit("ODT1_CMD_Hand")
      Appearance <- "ODT1_CMD_Hand"
      ProcessValue <- "ODT1_CMD_Hand"
   Button "Button_8" at 240,93 size 49x22; TextOff 'Выкл'
      on Click: ResetBit("ODT1_CMD_Start_M")
   Button "Button_9" at 184,93 size 47x22; TextOff 'Вкл'
      on Click: SetBit("ODT1_CMD_Start_M")
      Appearance <- "ODT1_CMD_Start_M"
   Button "Button_10" at 360,70 size 46x20; TextOff 'Inv'
      on Click: InvertBit("ODT1_CMD_Inverse")
      Appearance <- "ODT1_CMD_Inverse"
   Button "Button_11" at 360,95 size 46x20; TextOff 'Sim'
      on Click: InvertBit("ODT1_CMD_Simulation")
      Appearance <- "ODT1_CMD_Simulation"
   TextField "Text field_3" at 131,11 size 45x22; Text 'Q 2.0'
   TextField "Text field_4" at 176,11 size 62x22; Text 'T0 CMD'
   Circle "Circle_3" at 131,34 size 22x22
      Appearance <- "ODT0_CMD_Start_A"
   Circle "Circle_4" at 154,34 size 22x22
      Appearance <- "ODT0_CMD_Q"
   Button "Button_12" at 298,12 size 59x44; TextOff 'Авто'; TextList "Hand"
      on Click: InvertBit("ODT0_CMD_Hand")
      Appearance <- "ODT0_CMD_Hand"
      ProcessValue <- "ODT0_CMD_Hand"
   Button "Button_13" at 240,34 size 49x22; TextOff 'Выкл'
      on Click: ResetBit("ODT0_CMD_Start_M")
   Button "Button_14" at 184,34 size 47x22; TextOff 'Вкл'
      on Click: SetBit("ODT0_CMD_Start_M")
      Appearance <- "ODT0_CMD_Start_M"
   Button "Button_15" at 360,11 size 46x20; TextOff 'Inv'
      on Click: InvertBit("ODT0_CMD_Inverse")
      Appearance <- "ODT0_CMD_Inverse"
   Button "Button_16" at 360,36 size 46x20; TextOff 'Sim'
      on Click: InvertBit("ODT0_CMD_Simulation")
      Appearance <- "ODT0_CMD_Simulation"
   TextField "Text field_5" at 131,129 size 45x22; Text 'Q 2.1'
   TextField "Text field_6" at 176,129 size 62x22; Text 'T2 CMD'
   Circle "Circle_5" at 131,152 size 22x22
      Appearance <- "ODT2_CMD_Start_A"
   Circle "Circle_6" at 154,152 size 22x22
      Appearance <- "ODT2_CMD_Q"
   Button "Button_17" at 298,130 size 59x44; TextOff 'Авто'; TextList "Hand"
      on Click: InvertBit("ODT2_CMD_Hand")
      Appearance <- "ODT2_CMD_Hand"
      ProcessValue <- "ODT2_CMD_Hand"
   Button "Button_18" at 240,152 size 49x22; TextOff 'Выкл'
      on Click: ResetBit("ODT2_CMD_Start_M")
   Button "Button_19" at 184,152 size 47x22; TextOff 'Вкл'
      on Click: SetBit("ODT2_CMD_Start_M")
      Appearance <- "ODT2_CMD_Start_M"
   Button "Button_20" at 360,129 size 46x20; TextOff 'Inv'
      on Click: InvertBit("ODT2_CMD_Inverse")
      Appearance <- "ODT2_CMD_Inverse"
   Button "Button_21" at 360,154 size 46x20; TextOff 'Sim'
      on Click: InvertBit("ODT2_CMD_Simulation")
      Appearance <- "ODT2_CMD_Simulation"
   TextField "Text field_7" at 131,188 size 45x22; Text 'Q 2.1'
   TextField "Text field_8" at 176,188 size 62x22; Text 'T3 CMD'
   Circle "Circle_7" at 131,211 size 22x22
      Appearance <- "ODT3_CMD_Start_A"
   Circle "Circle_8" at 154,211 size 22x22
      Appearance <- "ODT3_CMD_Q"
   Button "Button_22" at 298,189 size 59x44; TextOff 'Авто'; TextList "Hand"
      on Click: InvertBit("ODT3_CMD_Hand")
      Appearance <- "ODT3_CMD_Hand"
      ProcessValue <- "ODT3_CMD_Hand"
   Button "Button_23" at 240,211 size 49x22; TextOff 'Выкл'
      on Click: ResetBit("ODT3_CMD_Start_M")
   Button "Button_24" at 184,211 size 47x22; TextOff 'Вкл'
      on Click: SetBit("ODT3_CMD_Start_M")
      Appearance <- "ODT3_CMD_Start_M"
   Button "Button_25" at 360,188 size 46x20; TextOff 'Inv'
      on Click: InvertBit("ODT3_CMD_Inverse")
      Appearance <- "ODT3_CMD_Inverse"
   Button "Button_26" at 360,213 size 46x20; TextOff 'Sim'
      on Click: InvertBit("ODT3_CMD_Simulation")
      Appearance <- "ODT3_CMD_Simulation"
   Button "Button_1" at 7,5 size 96x32; TextOff 'Коробки'; Authorization "Admin"
      on Release: ActivateScreen("Conveyors_0", 0); SetTag("settings", 1)
      Appearance <- "settings"
   Button "Button_2" at 7,51 size 96x32; TextOff 'Шоколад'; Authorization "Admin"
      on Release: ActivateScreen("Conveyors_1", 0); SetTag("settings", 2)
      Appearance <- "settings"
   Button "Button_3" at 7,98 size 96x32; TextOff 'Клапана'; Authorization "Admin"
      on Release: SetTag("settings", 3); ActivateScreen("Valve", 0)
      Appearance <- "settings"
   Button "Button_4" at 7,145 size 96x32; TextOff 'DI 1'; Authorization "Admin"
      on Release: SetTag("settings", 4); ActivateScreen("DI_1", 0)
      Appearance <- "settings"
   Button "Button_5" at 7,191 size 96x32; TextOff 'DI 2'; Authorization "Admin"
      on Release: SetTag("settings", 5); ActivateScreen("DI_2", 0)
      Appearance <- "settings"
   Button "Button_6" at 7,238 size 96x32; TextOff 'DO'; Authorization "Admin"
      on Release: SetTag("settings", 6); ActivateScreen("DO", 0)
      Appearance <- "settings"
   Button "Button_77" at 7,285 size 96x32; TextOff 'Весы'; Authorization "Admin"
      on Press: ActivateScreen("0.0.0_Service_Quick_Start", 0)
      Appearance <- "settings"

screen "DI_2" 800x480, template "Main"
   TextField "Text field_7" at 131,187 size 45x22; Text 'I 2.3'
   TextField "Text field_8" at 176,187 size 88x22; Text 'К3 открыт'
   Circle "Circle_7" at 131,210 size 22x22
      Appearance <- "FB_K3_Open_Input"
   Circle "Circle_8" at 154,210 size 22x22
      Appearance <- "FB_K3_Open_Signal"
   Button "Button_19" at 298,188 size 59x44; TextOff 'Авто'; TextList "Hand"
      on Click: InvertBit("FB_K3_Open_Hand")
      Appearance <- "FB_K3_Open_Hand"
      ProcessValue <- "FB_K3_Open_Hand"
   Button "Button_20" at 240,210 size 49x22; TextOff 'Выкл'
      on Click: ResetBit("FB_K3_Open_Start_M")
   Button "Button_21" at 184,210 size 47x22; TextOff 'Вкл'
      on Click: SetBit("FB_K3_Open_Start_M")
      Appearance <- "FB_K3_Open_Start_M"
   IOField "I/O field_5" at 360,210 size 23x22; FormatPattern 99
      ProcessValue <- "FB_K3_Open_Filter_On_SP"
   IOField "I/O field_8" at 383,210 size 23x22; FormatPattern 99
      ProcessValue <- "FB_K3_Open_Filter_Off_SP"
   Button "Button_22" at 360,187 size 46x20; TextOff 'Inv'
      on Click: InvertBit("FB_K3_Open_Inverse")
      Appearance <- "FB_K3_Open_Inverse"
   TextField "Text field_5" at 131,128 size 45x22; Text 'I 2.2'
   TextField "Text field_6" at 176,128 size 87x22; Text 'К2 закрыт'
   Circle "Circle_5" at 131,151 size 22x22
      Appearance <- "FB_K2_Close_Input"
   Circle "Circle_6" at 154,151 size 22x22
      Appearance <- "FB_K2_Close_Signal"
   Button "Button_15" at 298,129 size 59x44; TextOff 'Авто'; TextList "Hand"
      on Click: InvertBit("FB_K2_Close_Hand")
      Appearance <- "FB_K2_Close_Hand"
      ProcessValue <- "FB_K2_Close_Hand"
   Button "Button_16" at 240,151 size 49x22; TextOff 'Выкл'
      on Click: ResetBit("FB_K2_Close_Start_M")
   Button "Button_17" at 184,151 size 47x22; TextOff 'Вкл'
      on Click: SetBit("FB_K2_Close_Start_M")
      Appearance <- "FB_K2_Close_Start_M"
   IOField "I/O field_3" at 360,151 size 23x22; FormatPattern 99
      ProcessValue <- "FB_K2_Close_Filter_On_SP"
   IOField "I/O field_4" at 383,151 size 23x22; FormatPattern 99
      ProcessValue <- "FB_K2_Close_Filter_Off_SP"
   Button "Button_18" at 360,128 size 46x20; TextOff 'Inv'
      on Click: InvertBit("FB_K2_Close_Inverse")
      Appearance <- "FB_K2_Close_Inverse"
   TextField "Text field_3" at 131,69 size 45x22; Text 'I 2.1'
   TextField "Text field_4" at 176,69 size 88x22; Text 'К2 открыт'
   Circle "Circle_3" at 131,92 size 22x22
      Appearance <- "FB_K2_Open_Input"
   Circle "Circle_4" at 154,92 size 22x22
      Appearance <- "FB_K2_Open_Signal"
   Button "Button_10" at 298,70 size 59x44; TextOff 'Авто'; TextList "Hand"
      on Click: InvertBit("FB_K2_Open_Hand")
      Appearance <- "FB_K2_Open_Hand"
      ProcessValue <- "FB_K2_Open_Hand"
   Button "Button_11" at 240,92 size 49x22; TextOff 'Выкл'
      on Click: ResetBit("FB_K2_Open_Start_M")
   Button "Button_13" at 184,92 size 47x22; TextOff 'Вкл'
      on Click: SetBit("FB_K2_Open_Start_M")
      Appearance <- "FB_K2_Open_Start_M"
   IOField "I/O field_1" at 360,92 size 23x22; FormatPattern 99
      ProcessValue <- "FB_K2_Open_Filter_On_SP"
   IOField "I/O field_2" at 383,92 size 23x22; FormatPattern 99
      ProcessValue <- "FB_K2_Open_Filter_Off_SP"
   Button "Button_14" at 360,69 size 46x20; TextOff 'Inv'
      on Click: InvertBit("FB_K2_Open_Inverse")
      Appearance <- "FB_K2_Open_Inverse"
   TextField "Text field_1" at 131,10 size 45x22; Text 'I 2.0'
   TextField "Text field_2" at 176,10 size 88x22; Text 'К1 открыт'
   Circle "Circle_1" at 131,33 size 22x22
      Appearance <- "FB_K1_Close_Input"
   Circle "Circle_2" at 154,33 size 22x22
      Appearance <- "FB_K1_Close_Signal"
   Button "Button_7" at 298,11 size 59x44; TextOff 'Авто'; TextList "Hand"
      on Click: InvertBit("FB_K1_Close_Hand")
      Appearance <- "FB_K1_Close_Hand"
      ProcessValue <- "FB_K1_Close_Hand"
   Button "Button_8" at 240,33 size 49x22; TextOff 'Выкл'
      on Click: ResetBit("FB_K1_Close_Start_M")
   Button "Button_12" at 184,33 size 47x22; TextOff 'Вкл'
      on Click: SetBit("FB_K1_Close_Start_M")
      Appearance <- "FB_K1_Close_Start_M"
   IOField "I/O field_6" at 360,33 size 23x22; FormatPattern 99
      ProcessValue <- "FB_K1_Close_Filter_On_SP"
   IOField "I/O field_7" at 383,33 size 23x22; FormatPattern 99
      ProcessValue <- "FB_K1_Close_Filter_Off_SP"
   Button "Button_9" at 360,10 size 46x20; TextOff 'Inv'
      on Click: InvertBit("FB_K1_Close_Inverse")
      Appearance <- "FB_K1_Close_Inverse"
   TextField "Text field_9" at 131,247 size 45x22; Text 'I 2.4'
   TextField "Text field_10" at 176,247 size 87x22; Text 'К3 закрыт'
   Circle "Circle_9" at 131,270 size 22x22
      Appearance <- "FB_K3_Close_Input"
   Circle "Circle_10" at 154,270 size 22x22
      Appearance <- "FB_K3_Close_Signal"
   Button "Button_23" at 298,248 size 59x44; TextOff 'Авто'; TextList "Hand"
      on Click: InvertBit("FB_K3_Close_Hand")
      Appearance <- "FB_K3_Close_Hand"
      ProcessValue <- "FB_K3_Close_Hand"
   Button "Button_24" at 240,270 size 49x22; TextOff 'Выкл'
      on Click: ResetBit("FB_K3_Close_Start_M")
   Button "Button_25" at 184,270 size 47x22; TextOff 'Вкл'
      on Click: SetBit("FB_K3_Close_Start_M")
      Appearance <- "FB_K3_Close_Start_M"
   IOField "I/O field_9" at 360,270 size 23x22; FormatPattern 99
      ProcessValue <- "FB_K3_Close_Filter_On_SP"
   IOField "I/O field_10" at 383,270 size 23x22; FormatPattern 99
      ProcessValue <- "FB_K3_Close_Filter_Off_SP"
   Button "Button_26" at 360,247 size 46x20; TextOff 'Inv'
      on Click: InvertBit("FB_K3_Close_Inverse")
      Appearance <- "FB_K3_Close_Inverse"
   Button "Button_1" at 7,5 size 96x32; TextOff 'Коробки'; Authorization "Admin"
      on Release: ActivateScreen("Conveyors_0", 0); SetTag("settings", 1)
      Appearance <- "settings"
   Button "Button_2" at 7,51 size 96x32; TextOff 'Шоколад'; Authorization "Admin"
      on Release: ActivateScreen("Conveyors_1", 0); SetTag("settings", 2)
      Appearance <- "settings"
   Button "Button_3" at 7,98 size 96x32; TextOff 'Клапана'; Authorization "Admin"
      on Release: SetTag("settings", 3); ActivateScreen("Valve", 0)
      Appearance <- "settings"
   Button "Button_4" at 7,145 size 96x32; TextOff 'DI 1'; Authorization "Admin"
      on Release: SetTag("settings", 4); ActivateScreen("DI_1", 0)
      Appearance <- "settings"
   Button "Button_5" at 7,191 size 96x32; TextOff 'DI 2'; Authorization "Admin"
      on Release: SetTag("settings", 5); ActivateScreen("DI_2", 0)
      Appearance <- "settings"
   Button "Button_6" at 7,238 size 96x32; TextOff 'DO'; Authorization "Admin"
      on Release: SetTag("settings", 6); ActivateScreen("DO", 0)
      Appearance <- "settings"
   Button "Button_27" at 7,285 size 96x32; TextOff 'Весы'; Authorization "Admin"
      on Press: ActivateScreen("0.0.0_Service_Quick_Start", 0)
      Appearance <- "settings"

screen "Memory" 800x480, template "Main"
   IOField "I/O field_13" at 381,77 size 347x30; FormatPattern ??????????????????????
      ProcessValue <- "T3V3W3_DB_part_names{12}"
   IOField "I/O field_14" at 381,114 size 347x30; FormatPattern ??????????????????????
      ProcessValue <- "T3V3W3_DB_part_names{13}"
   IOField "I/O field_15" at 381,150 size 347x30; FormatPattern ??????????????????????
      ProcessValue <- "T3V3W3_DB_part_names{14}"
   IOField "I/O field_16" at 381,185 size 347x30; FormatPattern ??????????????????????
      ProcessValue <- "T3V3W3_DB_part_names{15}"
   IOField "I/O field_17" at 381,222 size 347x30; FormatPattern ??????????????????????
      ProcessValue <- "T3V3W3_DB_part_names{16}"
   IOField "I/O field_18" at 381,259 size 347x30; FormatPattern ??????????????????????
      ProcessValue <- "T3V3W3_DB_part_names{17}"
   IOField "I/O field_19" at 381,294 size 347x30; FormatPattern ??????????????????????
      ProcessValue <- "T3V3W3_DB_part_names{18}"
   IOField "I/O field_20" at 381,331 size 347x30; FormatPattern ??????????????????????
      ProcessValue <- "T3V3W3_DB_part_names{19}"
   IOField "I/O field_12" at 381,41 size 347x30; FormatPattern ??????????????????????
      ProcessValue <- "T3V3W3_DB_part_names{11}"
   IOField "I/O field_11" at 381,5 size 347x30; FormatPattern ??????????????????????
      ProcessValue <- "T3V3W3_DB_part_names{10}"
   IOField "I/O field_3" at 10,77 size 347x30; FormatPattern ??????????????????????
      ProcessValue <- "T3V3W3_DB_part_names{2}"
   IOField "I/O field_4" at 10,114 size 347x30; FormatPattern ??????????????????????
      ProcessValue <- "T3V3W3_DB_part_names{3}"
   IOField "I/O field_5" at 10,150 size 347x30; FormatPattern ??????????????????????
      ProcessValue <- "T3V3W3_DB_part_names{4}"
   IOField "I/O field_6" at 10,185 size 347x30; FormatPattern ??????????????????????
      ProcessValue <- "T3V3W3_DB_part_names{5}"
   IOField "I/O field_7" at 10,222 size 347x30; FormatPattern ??????????????????????
      ProcessValue <- "T3V3W3_DB_part_names{6}"
   IOField "I/O field_8" at 10,259 size 347x30; FormatPattern ??????????????????????
      ProcessValue <- "T3V3W3_DB_part_names{7}"
   IOField "I/O field_9" at 10,294 size 347x30; FormatPattern ??????????????????????
      ProcessValue <- "T3V3W3_DB_part_names{8}"
   IOField "I/O field_10" at 10,331 size 347x30; FormatPattern ??????????????????????
      ProcessValue <- "T3V3W3_DB_part_names{9}"
   IOField "I/O field_2" at 10,41 size 347x30; FormatPattern ??????????????????????
      ProcessValue <- "T3V3W3_DB_part_names{1}"
   IOField "I/O field_1" at 10,5 size 347x30; FormatPattern ??????????????????????
      ProcessValue <- "T3V3W3_DB_part_names{0}"
   Button "Button_5" at 14,415 size 211x58; TextOff 'Обзор'
      on Click: ActivateScreen("Root screen", 0); SetTag("main_screens", 0)
      Appearance <- "main_screens"
   Button "Button_1" at 264,415 size 211x58; TextOff 'Вес'
      on Click: ActivateScreen("weight", 0); SetTag("main_screens", 1)
      Appearance <- "main_screens"
   Button "Button_2" at 513,415 size 211x58; TextOff 'Статистика'
      on Click: ActivateScreen("statistic", 0); SetTag("main_screens", 2); SetTag("stat_view", 0)
      Appearance <- "main_screens"
   Button "Button_3" at 150,363 size 211x46; TextOff 'Данные'
      on Click: ActivateScreen("statistic", 0); SetTag("stat_view", 0)
      Appearance <- "stat_view"
   Button "Button_9" at 372,363 size 211x46; TextOff 'Память'
      on Click: ActivateScreen("Memory", 0); SetTag("stat_view", 1)
      Appearance <- "stat_view"
   Button "Button_10" at 269,8 size 84x23; TextOff 'Удалить'
      on Click: SetBit("del_stat_mem_DB_del"); SetTag("del_stat_mem_DB_number", 0)
   Button "Button_7" at 269,44 size 84x23; TextOff 'Удалить'
      on Click: SetBit("del_stat_mem_DB_del"); SetTag("del_stat_mem_DB_number", 1)
   Button "Button_8" at 269,80 size 84x23; TextOff 'Удалить'
      on Click: SetBit("del_stat_mem_DB_del"); SetTag("del_stat_mem_DB_number", 2)
   Button "Button_11" at 269,117 size 84x23; TextOff 'Удалить'
      on Click: SetBit("del_stat_mem_DB_del"); SetTag("del_stat_mem_DB_number", 3)
   Button "Button_12" at 269,153 size 84x23; TextOff 'Удалить'
      on Click: SetBit("del_stat_mem_DB_del"); SetTag("del_stat_mem_DB_number", 4)
   Button "Button_13" at 269,189 size 84x23; TextOff 'Удалить'
      on Click: SetBit("del_stat_mem_DB_del"); SetTag("del_stat_mem_DB_number", 5)
   Button "Button_14" at 269,225 size 84x23; TextOff 'Удалить'
      on Click: SetBit("del_stat_mem_DB_del"); SetTag("del_stat_mem_DB_number", 6)
   Button "Button_15" at 269,262 size 84x23; TextOff 'Удалить'
      on Click: SetBit("del_stat_mem_DB_del"); SetTag("del_stat_mem_DB_number", 7)
   Button "Button_16" at 269,297 size 84x23; TextOff 'Удалить'
      on Click: SetBit("del_stat_mem_DB_del"); SetTag("del_stat_mem_DB_number", 8)
   Button "Button_17" at 269,334 size 84x23; TextOff 'Удалить'
      on Click: SetBit("del_stat_mem_DB_del"); SetTag("del_stat_mem_DB_number", 9)
   Button "Button_18" at 640,8 size 84x23; TextOff 'Удалить'
      on Click: SetBit("del_stat_mem_DB_del"); SetTag("del_stat_mem_DB_number", 10)
   Button "Button_19" at 640,44 size 84x23; TextOff 'Удалить'
      on Click: SetBit("del_stat_mem_DB_del"); SetTag("del_stat_mem_DB_number", 11)
   Button "Button_20" at 640,80 size 84x23; TextOff 'Удалить'
      on Click: SetBit("del_stat_mem_DB_del"); SetTag("del_stat_mem_DB_number", 12)
   Button "Button_21" at 640,117 size 84x23; TextOff 'Удалить'
      on Click: SetBit("del_stat_mem_DB_del"); SetTag("del_stat_mem_DB_number", 13)
   Button "Button_22" at 640,153 size 84x23; TextOff 'Удалить'
      on Click: SetBit("del_stat_mem_DB_del"); SetTag("del_stat_mem_DB_number", 14)
   Button "Button_23" at 640,188 size 84x23; TextOff 'Удалить'
      on Click: SetBit("del_stat_mem_DB_del"); SetTag("del_stat_mem_DB_number", 15)
   Button "Button_24" at 640,225 size 84x23; TextOff 'Удалить'
      on Click: SetBit("del_stat_mem_DB_del"); SetTag("del_stat_mem_DB_number", 16)
   Button "Button_25" at 640,262 size 84x23; TextOff 'Удалить'
      on Click: SetBit("del_stat_mem_DB_del"); SetTag("del_stat_mem_DB_number", 17)
   Button "Button_26" at 640,297 size 84x23; TextOff 'Удалить'
      on Click: SetBit("del_stat_mem_DB_del"); SetTag("del_stat_mem_DB_number", 18)
   Button "Button_27" at 640,334 size 84x23; TextOff 'Удалить'
      on Click: SetBit("del_stat_mem_DB_del"); SetTag("del_stat_mem_DB_number", 19)

screen "Alarms" 800x480, template "Main"
   AlarmView "Alarm view_1" at 4,3 size 718x470; ColumnTextDate 'Дата'; ColumnTextAlarmState 'Статус'; ColumnTextTime 'Время'; ColumnTextAlarmText 'Аварийное сообщение'

screen "Calibration" 800x480, template "Main"
   TextField "Text field_1" at 256,5 size 233x47; Text 'Калибровка'

screen "SP" 800x480, template "Main"
   TextField "Text field_1" at 288,5 size 156x47; Text 'Уставки'
   GraphicView "Graphic view_5" at 367,50 size 347x209; Picture "clean2"
   TextField "Text field_21" at 485,64 size 112x33; Text 'Дозация'
   TextField "Text field_22" at 380,118 size 122x23; Text 'Уставка веса:'
   TextField "Text field_23" at 666,118 size 43x23; Text 'кг'
   GraphicView "Graphic view_6" at 598,113 size 66x33; Picture "input_1"
   IOField "I/O field_3" at 602,116 size 58x27; Authorization "Operator"; FormatPattern 99.9
      ProcessValue <- "T3V3W3_DB_SetPoints_SP"
   TextField "Text field_24" at 380,152 size 201x23; Text 'Уставка веса в полете:'
   TextField "Text field_25" at 667,152 size 43x23; Text 'кг'
   GraphicView "Graphic view_7" at 598,149 size 66x33; Picture "input_1"
   IOField "I/O field_9" at 602,152 size 58x27; Authorization "Operator"; FormatPattern 9.999
      ProcessValue <- "T3V3W3_DB_SetPoints_SP_fly"
   GraphicView "Graphic view_14" at 598,183 size 66x33; Picture "input_1"
   TextField "Text field_30" at 668,186 size 43x23; Text 'кг'
   IOField "I/O field_10" at 602,186 size 58x27; Authorization "Operator"; FormatPattern 9.999
      ProcessValue <- "T3V3W3_DB_SetPoints_delta_add"
   TextField "Text field_29" at 380,186 size 170x23; Text 'Откл. от уставки +:'
   GraphicView "Graphic view_1" at 20,50 size 347x209; Picture "clean2"
   TextField "Text field_2" at 135,64 size 117x33; Text 'Таймеры'
   TextField "Text field_31" at 35,118 size 199x23; Text 'Балансировка веса до:'
   TextField "Text field_32" at 321,118 size 43x23; Text 'с'
   GraphicView "Graphic view_15" at 253,113 size 66x33; Picture "input_1"
   GraphicView "Graphic view_8" at 598,217 size 66x33; Picture "input_1"
   TextField "Text field_9" at 668,220 size 43x23; Text 'кг'
   TextField "Text field_10" at 380,220 size 164x23; Text 'Откл. от уставки -:'
   IOField "I/O field_5" at 257,116 size 58x27; Authorization "Operator"; FormatPattern 999.99
      ProcessValue <- "T3V3W3_DB_Timers_T_s7_SP"
   TextField "Text field_12" at 35,152 size 191x23; Text 'Балансир. веса после:'
   TextField "Text field_13" at 321,152 size 43x23; Text 'с'
   GraphicView "Graphic view_10" at 253,149 size 66x33; Picture "input_1"
   TextField "Text field_17" at 321,186 size 43x23; Text 'с'
   GraphicView "Graphic view_12" at 253,183 size 66x33; Picture "input_1"
   IOField "I/O field_7" at 257,152 size 58x27; Authorization "Operator"; FormatPattern 999.99
      ProcessValue <- "T3V3W3_DB_Timers_T_s15_SP"
   IOField "I/O field_11" at 602,220 size 58x27; Authorization "Operator"; FormatPattern 9.999
      ProcessValue <- "T3V3W3_DB_SetPoints_delata_sub"
   TextField "Text field_3" at 35,186 size 172x23; Text 'Время на упаковку:'
   IOField "I/O field_1" at 257,186 size 58x27; Authorization "Operator"; FormatPattern 999.99
      ProcessValue <- "T4D4_S2_SP"
   GraphicView "Graphic view_3" at 20,261 size 347x209; Picture "clean2"
   TextField "Text field_5" at 138,275 size 112x33; Text 'Дозация'
   TextField "Text field_18" at 33,320 size 272x23; Text 'Переход на малую скорость за:'
   TextField "Text field_19" at 319,351 size 43x23; Text 'кг'
   GraphicView "Graphic view_13" at 251,346 size 66x33; Picture "input_1"
   IOField "I/O field_2" at 255,349 size 58x27; Authorization "Operator"; FormatPattern 99.9
      ProcessValue <- "T3V3W3_DB_SetPoints_SP_ch_s"
   TextField "Text field_6" at 321,383 size 43x23; Text '%'
   TextField "Text field_20" at 33,383 size 213x23; Text 'Максимальная скорость:'
   GraphicView "Graphic view_16" at 251,414 size 66x33; Picture "input_1"
   TextField "Text field_26" at 321,417 size 43x23; Text '%'
   TextField "Text field_27" at 33,417 size 205x23; Text 'Минимальная скорость:'
   GraphicView "Graphic view_17" at 251,380 size 66x33; Picture "input_1"
   IOField "I/O field_13" at 255,417 size 58x27; Authorization "Operator"; FormatPattern 999.9
      ProcessValue <- "T0T1_DB_SP_min"
   IOField "I/O field_12" at 255,383 size 58x27; Authorization "Operator"; FormatPattern 999.9
      ProcessValue <- "T0T1_DB_SP_max"

screen "Monitor" 800x480, template "Main"
   TextField "Text field_1" at 168,4 size 424x47; Text 'Параметры установки'
   Button "Button_1" at 7,5 size 96x32; TextOff 'Коробки'; Authorization "Admin"
      on Release: ActivateScreen("Conveyors_0", 0); SetTag("settings", 1)
      Appearance <- "settings"
   Button "Button_2" at 7,51 size 96x32; TextOff 'Шоколад'; Authorization "Admin"
      on Release: ActivateScreen("Conveyors_1", 0); SetTag("settings", 2)
      Appearance <- "settings"
   Button "Button_3" at 7,98 size 96x32; TextOff 'Клапана'; Authorization "Admin"
      on Release: SetTag("settings", 3); ActivateScreen("Valve", 0)
      Appearance <- "settings"
   Button "Button_4" at 7,145 size 96x32; TextOff 'DI 1'; Authorization "Admin"
      on Release: SetTag("settings", 4); ActivateScreen("DI_1", 0)
      Appearance <- "settings"
   Button "Button_5" at 7,191 size 96x32; TextOff 'DI 2'; Authorization "Admin"
      on Release: SetTag("settings", 5); ActivateScreen("DI_2", 0)
      Appearance <- "settings"
   Button "Button_6" at 7,238 size 96x32; TextOff 'DO'; Authorization "Admin"
      on Release: SetTag("settings", 6); ActivateScreen("DO", 0)
      Appearance <- "settings"
   GraphicView "Graphic view_1" at 123,52 size 347x209; Picture "clean2"
   TextField "Text field_2" at 263,66 size 68x33; Text 'Весы'
   TextField "Text field_4" at 424,120 size 43x23; Text 'кг'
   GraphicView "Graphic view_2" at 356,115 size 66x33; Picture "input_1"
   TextField "Text field_7" at 138,154 size 93x23; Text 'Поправка:'
   TextField "Text field_8" at 424,154 size 43x23; Text 'кг'
   GraphicView "Graphic view_4" at 356,151 size 66x33; Picture "input_1"
   IOField "I/O field_4" at 360,154 size 58x27; Authorization "Operator"; FormatPattern s99.99
      ProcessValue <- "T3V3W3_DB_LocalVar_Sp_start"
   TextField "Text field_16" at 138,119 size 120x23; Text 'Текущий вес:'
   IOField "I/O field_6" at 360,118 size 58x27; Authorization "Operator"; FormatPattern 99.99
      ProcessValue <- "T3V3W3_DB_LocalVar_SP_loaded"
   Button "Button_7" at 200,198 size 193x44; TextOff 'Установка нуля'; TextList "Hand"
      on Click: InvertBit("T3V3W3_DB_Reset_weight")
      ProcessValue <- "ODT1_CMD_Hand"
   Button "Button_8" at 7,285 size 96x32; TextOff 'Весы'; Authorization "Admin"
      Appearance <- "settings"
      on Press: ActivateScreen("0.0.0_Service_Quick_Start", 0)

screen "weight" 800x480, template "Main"
   IOField "I/O field_2" at 14,15 size 714x396; FormatPattern s99.99
      ProcessValue <- "T3V3W3_DB_LocalVar_SP_loaded"
   Button "Button_16" at 15,17 size 713x392; TextOff 'Установка нуля'; TextList "Hand"
      on Click: InvertBit("T3V3W3_DB_Reset_weight")
      ProcessValue <- "ODT1_CMD_Hand"
      Visibility <- "Logic_DB_Start_weight"
   Button "Button_5" at 14,415 size 211x58; TextOff 'Обзор'
      on Click: ActivateScreen("Root screen", 0); SetTag("main_screens", 0)
      Appearance <- "main_screens"
   Button "Button_14" at 264,415 size 211x58; TextOff 'Вес'
      on Click: ActivateScreen("weight", 0); SetTag("main_screens", 1)
      Appearance <- "main_screens"
   Button "Button_7" at 513,415 size 211x58; TextOff 'Статистика'
      on Click: ActivateScreen("statistic", 0); SetTag("main_screens", 2); SetTag("stat_view", 0)
      Appearance <- "main_screens"
   Button "Button_15" at 13,357 size 178x54; TextOff 'Пропустить'
      on Click: SetBit("T3V3W3_DB_Skip_box")
      Appearance <- "main_screens"
   Rectangle "Rectangle_33" at 21,1 size 715x106
      Visibility <- "T3V3W3_DB_Reload"
   TextField "Text field_5" at 151,19 size 455x58; Text 'Некорректный вес.'
      Visibility <- "T3V3W3_DB_Reload"
   Button "Button_1" at 206,316 size 345x75; TextOff 'Продолжить'
      on Click: SetBit("Reset_All")
      Visibility <- "T3V3W3_DB_Reload"
   Rectangle "Rectangle_34" at 21,15 size 714x90
      Visibility <- "T3V3W3_DB_No_box"
   Button "Button_20" at 217,305 size 345x75; TextOff 'Продолжить'
      on Click: ResetBit("T3V3W3_DB_No_box")
      Visibility <- "T3V3W3_DB_No_box"
   TextField "Text field_6" at 223,32 size 311x58; Text 'Нет коробки.'
      Visibility <- "T3V3W3_DB_No_box"

